  LIN {X 1499.916,Y -481.788,Z -133.994,A 92.55766,B 0.00000,C 180.00000} ; insert
  LIN {X 1499.916,Y -481.788,Z -133.994,A 92.55766,B 0.00000,C 180.00000} ; release
  LIN {X 1499.916,Y -481.788,Z 166.006,A 92.55766,B 0.00000,C 180.00000} ; retreat
  ; Step 2458, bar 2905
  LIN {X 2249.916,Y -481.788,Z 1074.491,A 92.55766,B 0.00000,C 180.00000} ; outside
  LIN {X 2249.916,Y -481.788,Z 116.006,A 92.55766,B 0.00000,C 180.00000} ; preinsert
  LIN {X 2249.916,Y -481.788,Z -133.994,A 92.55766,B 0.00000,C 180.00000} ; insert
  LIN {X 2249.916,Y -481.788,Z -133.994,A 92.55766,B 0.00000,C 180.00000} ; release
  LIN {X 2249.916,Y -481.788,Z 166.006,A 92.55766,B 0.00000,C 180.00000} ; retreat
  ; Step 2459, bar 2908
  LIN {X 2999.916,Y -481.788,Z 1074.491,A 92.55766,B 0.00000,C 180.00000} ; outside
  LIN {X 2999.916,Y -481.788,Z 116.006,A 92.55766,B 0.00000,C 180.00000} ; preinsert
  LIN {X 2999.916,Y -481.788,Z -133.994,A 92.55766,B 0.00000,C 180.00000} ; insert
  LIN {X 2999.916,Y -481.788,Z -133.994,A 92.55766,B 0.00000,C 180.00000} ; release
  LIN {X 2999.916,Y -481.788,Z 166.006,A 92.55766,B 0.00000,C 180.00000} ; retreat
  ; Step 2460, bar 2911
  LIN {X 3749.916,Y -481.788,Z 1074.491,A 92.55766,B 0.00000,C 180.00000} ; outside
  LIN {X 3749.916,Y -481.788,Z 116.006,A 92.55766,B 0.00000,C 180.00000} ; preinsert
  LIN {X 3749.916,Y -481.788,Z -133.994,A 92.55766,B 0.00000,C 180.00000} ; insert
  LIN {X 3749.916,Y -481.788,Z -133.994,A 92.55766,B 0.00000,C 180.00000} ; release
  LIN {X 3749.916,Y -481.788,Z 166.006,A 92.55766,B 0.00000,C 180.00000} ; retreat
  ; Step 2461, bar 2914
  LIN {X 4499.916,Y -481.788,Z 1074.491,A 92.55766,B 0.00000,C 180.00000} ; outside
  LIN {X 4499.916,Y -481.788,Z 116.006,A 92.55766,B 0.00000,C 180.00000} ; preinsert
  LIN {X 4499.916,Y -481.788,Z -133.994,A 92.55766,B 0.00000,C 180.00000} ; insert
  LIN {X 4499.916,Y -481.788,Z -133.994,A 92.55766,B 0.00000,C 180.00000} ; release
  LIN {X 4499.916,Y -481.788,Z 166.006,A 92.55766,B 0.00000,C 180.00000} ; retreat
  ; Step 2462, bar 2917
  LIN {X 5249.916,Y -481.788,Z 1074.491,A 92.55766,B 0.00000,C 180.00000} ; outside
  LIN {X 5249.916,Y -481.788,Z 116.006,A 92.55766,B 0.00000,C 180.00000} ; preinsert
  LIN {X 5249.916,Y -481.788,Z -133.994,A 92.55766,B 0.00000,C 180.00000} ; insert
  LIN {X 5249.916,Y -481.788,Z -133.994,A 92.55766,B 0.00000,C 180.00000} ; release
  LIN {X 5249.916,Y -481.788,Z 166.006,A 92.55766,B 0.00000,C 180.00000} ; retreat
  ; Step 2463, bar 2920
  LIN {X 5999.916,Y -481.788,Z 1074.491,A 92.55766,B 0.00000,C 180.00000} ; outside
  LIN {X 5999.916,Y -481.788,Z 116.006,A 92.55766,B 0.00000,C 180.00000} ; preinsert
  LIN {X 5999.916,Y -481.788,Z -133.994,A 92.55766,B 0.00000,C 180.00000} ; insert
  LIN {X 5999.916,Y -481.788,Z -133.994,A 92.55766,B 0.00000,C 180.00000} ; release
  LIN {X 5999.916,Y -481.788,Z 166.006,A 92.55766,B 0.00000,C 180.00000} ; retreat
  ; Step 2464, bar 2923
  LIN {X 6749.916,Y -481.788,Z 1074.491,A 92.55766,B 0.00000,C 180.00000} ; outside
  LIN {X 6749.916,Y -481.788,Z 116.006,A 92.55766,B 0.00000,C 180.00000} ; preinsert
  LIN {X 6749.916,Y -481.788,Z -133.994,A 92.55766,B 0.00000,C 180.00000} ; insert
  LIN {X 6749.916,Y -481.788,Z -133.994,A 92.55766,B 0.00000,C 180.00000} ; release
  LIN {X 6749.916,Y -481.788,Z 166.006,A 92.55766,B 0.00000,C 180.00000} ; retreat
  ; Step 2465, bar 2926
  LIN {X 7499.916,Y -481.788,Z 1074.491,A 92.55766,B 0.00000,C 180.00000} ; outside
  LIN {X 7499.916,Y -481.788,Z 116.006,A 92.55766,B 0.00000,C 180.00000} ; preinsert
  LIN {X 7499.916,Y -481.788,Z -133.994,A 92.55766,B 0.00000,C 180.00000} ; insert
  LIN {X 7499.916,Y -481.788,Z -133.994,A 92.55766,B 0.00000,C 180.00000} ; release
  LIN {X 7499.916,Y -481.788,Z 166.006,A 92.55766,B 0.00000,C 180.00000} ; retreat
  ; Step 2466, bar 2929
  LIN {X 8249.916,Y -481.788,Z 1074.491,A 92.55766,B 0.00000,C 180.00000} ; outside
  LIN {X 8249.916,Y -481.788,Z 116.006,A 92.55766,B 0.00000,C 180.00000} ; preinsert
  LIN {X 8249.916,Y -481.788,Z -133.994,A 92.55766,B 0.00000,C 180.00000} ; insert
  LIN {X 8249.916,Y -481.788,Z -133.994,A 92.55766,B 0.00000,C 180.00000} ; release
  LIN {X 8249.916,Y -481.788,Z 166.006,A 92.55766,B 0.00000,C 180.00000} ; retreat
  ; Step 2467, bar 2932
  LIN {X 8999.916,Y -481.788,Z 1074.491,A 92.55766,B 0.00000,C 180.00000} ; outside
  LIN {X 8999.916,Y -481.788,Z 116.006,A 92.55766,B 0.00000,C 180.00000} ; preinsert
  LIN {X 8999.916,Y -481.788,Z -133.994,A 92.55766,B 0.00000,C 180.00000} ; insert
  LIN {X 8999.916,Y -481.788,Z -133.994,A 92.55766,B 0.00000,C 180.00000} ; release
  LIN {X 8999.916,Y -481.788,Z 166.006,A 92.55766,B 0.00000,C 180.00000} ; retreat
  ; Step 2468, bar 2935
  LIN {X 9749.916,Y -481.788,Z 1074.491,A 92.55766,B 0.00000,C 180.00000} ; outside
  LIN {X 9749.916,Y -481.788,Z 116.006,A 92.55766,B 0.00000,C 180.00000} ; preinsert
  LIN {X 9749.916,Y -481.788,Z -133.994,A 92.55766,B 0.00000,C 180.00000} ; insert
  LIN {X 9749.916,Y -481.788,Z -133.994,A 92.55766,B 0.00000,C 180.00000} ; release
  LIN {X 9749.916,Y -481.788,Z 166.006,A 92.55766,B 0.00000,C 180.00000} ; retreat
  ; Step 2469, bar 2938
  LIN {X 10499.916,Y -481.788,Z 1074.491,A 92.55766,B 0.00000,C 180.00000} ; outside
  LIN {X 10499.916,Y -481.788,Z 116.006,A 92.55766,B 0.00000,C 180.00000} ; preinsert
  LIN {X 10499.916,Y -481.788,Z -133.994,A 92.55766,B 0.00000,C 180.00000} ; insert
  LIN {X 10499.916,Y -481.788,Z -133.994,A 92.55766,B 0.00000,C 180.00000} ; release
  LIN {X 10499.916,Y -481.788,Z 166.006,A 92.55766,B 0.00000,C 180.00000} ; retreat
  ; Step 2470, bar 2941
  LIN {X 11249.916,Y -481.788,Z 1074.491,A 92.55766,B 0.00000,C 180.00000} ; outside
  LIN {X 11249.916,Y -481.788,Z 116.006,A 92.55766,B 0.00000,C 180.00000} ; preinsert
  LIN {X 11249.916,Y -481.788,Z -133.994,A 92.55766,B 0.00000,C 180.00000} ; insert
  LIN {X 11249.916,Y -481.788,Z -133.994,A 92.55766,B 0.00000,C 180.00000} ; release
  LIN {X 11249.916,Y -481.788,Z 166.006,A 92.55766,B 0.00000,C 180.00000} ; retreat
  ; Step 2471, bar 2943
  LIN {X 11999.916,Y -481.788,Z 1074.491,A 92.55766,B 0.00000,C 180.00000} ; outside
  LIN {X 11999.916,Y -481.788,Z 116.006,A 92.55766,B 0.00000,C 180.00000} ; preinsert
  LIN {X 11999.916,Y -481.788,Z -133.994,A 92.55766,B 0.00000,C 180.00000} ; insert
  LIN {X 11999.916,Y -481.788,Z -133.994,A 92.55766,B 0.00000,C 180.00000} ; release
  LIN {X 11999.916,Y -481.788,Z 166.006,A 92.55766,B 0.00000,C 180.00000} ; retreat
  ; Step 2472, bar 2636
  LIN {X -11999.916,Y 481.788,Z 1074.491,A -87.44234,B 0.00000,C 180.00000} ; outside
  LIN {X -11999.916,Y 481.788,Z 116.006,A -87.44234,B 0.00000,C 180.00000} ; preinsert
  LIN {X -11999.916,Y 481.788,Z -133.994,A -87.44234,B 0.00000,C 180.00000} ; insert
  LIN {X -11999.916,Y 481.788,Z -133.994,A -87.44234,B 0.00000,C 180.00000} ; release
  LIN {X -11999.916,Y 481.788,Z 166.006,A -87.44234,B 0.00000,C 180.00000} ; retreat
  ; Step 2473, bar 2631
  LIN {X -11249.916,Y 481.788,Z 1074.491,A -87.44234,B 0.00000,C 180.00000} ; outside
  LIN {X -11249.916,Y 481.788,Z 116.006,A -87.44234,B 0.00000,C 180.00000} ; preinsert
  LIN {X -11249.916,Y 481.788,Z -133.994,A -87.44234,B 0.00000,C 180.00000} ; insert
  LIN {X -11249.916,Y 481.788,Z -133.994,A -87.44234,B 0.00000,C 180.00000} ; release
  LIN {X -11249.916,Y 481.788,Z 166.006,A -87.44234,B 0.00000,C 180.00000} ; retreat
  ; Step 2474, bar 2624
  LIN {X -10499.916,Y 481.788,Z 1074.491,A -87.44234,B 0.00000,C 180.00000} ; outside
  LIN {X -10499.916,Y 481.788,Z 116.006,A -87.44234,B 0.00000,C 180.00000} ; preinsert
  LIN {X -10499.916,Y 481.788,Z -133.994,A -87.44234,B 0.00000,C 180.00000} ; insert
  LIN {X -10499.916,Y 481.788,Z -133.994,A -87.44234,B 0.00000,C 180.00000} ; release
  LIN {X -10499.916,Y 481.788,Z 166.006,A -87.44234,B 0.00000,C 180.00000} ; retreat
  ; Step 2475, bar 2617
  LIN {X -9749.916,Y 481.788,Z 1074.491,A -87.44234,B 0.00000,C 180.00000} ; outside
  LIN {X -9749.916,Y 481.788,Z 116.006,A -87.44234,B 0.00000,C 180.00000} ; preinsert
  LIN {X -9749.916,Y 481.788,Z -133.994,A -87.44234,B 0.00000,C 180.00000} ; insert
  LIN {X -9749.916,Y 481.788,Z -133.994,A -87.44234,B 0.00000,C 180.00000} ; release
  LIN {X -9749.916,Y 481.788,Z 166.006,A -87.44234,B 0.00000,C 180.00000} ; retreat
  ; Step 2476, bar 2610
  LIN {X -8999.916,Y 481.788,Z 1074.491,A -87.44234,B 0.00000,C 180.00000} ; outside
  LIN {X -8999.916,Y 481.788,Z 116.006,A -87.44234,B 0.00000,C 180.00000} ; preinsert
  LIN {X -8999.916,Y 481.788,Z -133.994,A -87.44234,B 0.00000,C 180.00000} ; insert
  LIN {X -8999.916,Y 481.788,Z -133.994,A -87.44234,B 0.00000,C 180.00000} ; release
  LIN {X -8999.916,Y 481.788,Z 166.006,A -87.44234,B 0.00000,C 180.00000} ; retreat
  ; Step 2477, bar 2603
  LIN {X -8249.916,Y 481.788,Z 1074.491,A -87.44234,B 0.00000,C 180.00000} ; outside
  LIN {X -8249.916,Y 481.788,Z 116.006,A -87.44234,B 0.00000,C 180.00000} ; preinsert
  LIN {X -8249.916,Y 481.788,Z -133.994,A -87.44234,B 0.00000,C 180.00000} ; insert
  LIN {X -8249.916,Y 481.788,Z -133.994,A -87.44234,B 0.00000,C 180.00000} ; release
  LIN {X -8249.916,Y 481.788,Z 166.006,A -87.44234,B 0.00000,C 180.00000} ; retreat
  ; Step 2478, bar 2596
  LIN {X -7499.916,Y 481.788,Z 1074.491,A -87.44234,B 0.00000,C 180.00000} ; outside
  LIN {X -7499.916,Y 481.788,Z 116.006,A -87.44234,B 0.00000,C 180.00000} ; preinsert
  LIN {X -7499.916,Y 481.788,Z -133.994,A -87.44234,B 0.00000,C 180.00000} ; insert
  LIN {X -7499.916,Y 481.788,Z -133.994,A -87.44234,B 0.00000,C 180.00000} ; release
  LIN {X -7499.916,Y 481.788,Z 166.006,A -87.44234,B 0.00000,C 180.00000} ; retreat
  ; Step 2479, bar 2589
  LIN {X -6749.916,Y 481.788,Z 1074.491,A -87.44234,B 0.00000,C 180.00000} ; outside
  LIN {X -6749.916,Y 481.788,Z 116.006,A -87.44234,B 0.00000,C 180.00000} ; preinsert
  LIN {X -6749.916,Y 481.788,Z -133.994,A -87.44234,B 0.00000,C 180.00000} ; insert
  LIN {X -6749.916,Y 481.788,Z -133.994,A -87.44234,B 0.00000,C 180.00000} ; release
  LIN {X -6749.916,Y 481.788,Z 166.006,A -87.44234,B 0.00000,C 180.00000} ; retreat
  ; Step 2480, bar 2582
  LIN {X -5999.916,Y 481.788,Z 1074.491,A -87.44234,B 0.00000,C 180.00000} ; outside
  LIN {X -5999.916,Y 481.788,Z 116.006,A -87.44234,B 0.00000,C 180.00000} ; preinsert
  LIN {X -5999.916,Y 481.788,Z -133.994,A -87.44234,B 0.00000,C 180.00000} ; insert
  LIN {X -5999.916,Y 481.788,Z -133.994,A -87.44234,B 0.00000,C 180.00000} ; release
  LIN {X -5999.916,Y 481.788,Z 166.006,A -87.44234,B 0.00000,C 180.00000} ; retreat
  ; Step 2481, bar 2575
  LIN {X -5249.916,Y 481.788,Z 1074.491,A -87.44234,B 0.00000,C 180.00000} ; outside
  LIN {X -5249.916,Y 481.788,Z 116.006,A -87.44234,B 0.00000,C 180.00000} ; preinsert
  LIN {X -5249.916,Y 481.788,Z -133.994,A -87.44234,B 0.00000,C 180.00000} ; insert
  LIN {X -5249.916,Y 481.788,Z -133.994,A -87.44234,B 0.00000,C 180.00000} ; release
  LIN {X -5249.916,Y 481.788,Z 166.006,A -87.44234,B 0.00000,C 180.00000} ; retreat
  ; Step 2482, bar 2568
  LIN {X -4499.916,Y 481.788,Z 1074.491,A -87.44234,B 0.00000,C 180.00000} ; outside
  LIN {X -4499.916,Y 481.788,Z 116.006,A -87.44234,B 0.00000,C 180.00000} ; preinsert
  LIN {X -4499.916,Y 481.788,Z -133.994,A -87.44234,B 0.00000,C 180.00000} ; insert
  LIN {X -4499.916,Y 481.788,Z -133.994,A -87.44234,B 0.00000,C 180.00000} ; release
  LIN {X -4499.916,Y 481.788,Z 166.006,A -87.44234,B 0.00000,C 180.00000} ; retreat
  ; Step 2483, bar 2561
  LIN {X -3749.916,Y 481.788,Z 1074.491,A -87.44234,B 0.00000,C 180.00000} ; outside
  LIN {X -3749.916,Y 481.788,Z 116.006,A -87.44234,B 0.00000,C 180.00000} ; preinsert
  LIN {X -3749.916,Y 481.788,Z -133.994,A -87.44234,B 0.00000,C 180.00000} ; insert
  LIN {X -3749.916,Y 481.788,Z -133.994,A -87.44234,B 0.00000,C 180.00000} ; release
  LIN {X -3749.916,Y 481.788,Z 166.006,A -87.44234,B 0.00000,C 180.00000} ; retreat
  ; Step 2484, bar 2554
  LIN {X -2999.916,Y 481.788,Z 1074.491,A -87.44234,B 0.00000,C 180.00000} ; outside
  LIN {X -2999.916,Y 481.788,Z 116.006,A -87.44234,B 0.00000,C 180.00000} ; preinsert
  LIN {X -2999.916,Y 481.788,Z -133.994,A -87.44234,B 0.00000,C 180.00000} ; insert
  LIN {X -2999.916,Y 481.788,Z -133.994,A -87.44234,B 0.00000,C 180.00000} ; release
  LIN {X -2999.916,Y 481.788,Z 166.006,A -87.44234,B 0.00000,C 180.00000} ; retreat
  ; Step 2485, bar 2547
  LIN {X -2249.916,Y 481.788,Z 1074.491,A -87.44234,B 0.00000,C 180.00000} ; outside
  LIN {X -2249.916,Y 481.788,Z 116.006,A -87.44234,B 0.00000,C 180.00000} ; preinsert
  LIN {X -2249.916,Y 481.788,Z -133.994,A -87.44234,B 0.00000,C 180.00000} ; insert
  LIN {X -2249.916,Y 481.788,Z -133.994,A -87.44234,B 0.00000,C 180.00000} ; release
  LIN {X -2249.916,Y 481.788,Z 166.006,A -87.44234,B 0.00000,C 180.00000} ; retreat
  ; Step 2486, bar 2540
  LIN {X -1499.916,Y 481.788,Z 1074.491,A -87.44234,B 0.00000,C 180.00000} ; outside
  LIN {X -1499.916,Y 481.788,Z 116.006,A -87.44234,B 0.00000,C 180.00000} ; preinsert
  LIN {X -1499.916,Y 481.788,Z -133.994,A -87.44234,B 0.00000,C 180.00000} ; insert
  LIN {X -1499.916,Y 481.788,Z -133.994,A -87.44234,B 0.00000,C 180.00000} ; release
  LIN {X -1499.916,Y 481.788,Z 166.006,A -87.44234,B 0.00000,C 180.00000} ; retreat
  ; Step 2487, bar 1974
  LIN {X 0.084,Y 481.788,Z 1074.491,A -87.44234,B 0.00000,C 180.00000} ; outside
  LIN {X 0.084,Y 481.788,Z 116.006,A -87.44234,B 0.00000,C 180.00000} ; preinsert
  LIN {X 0.084,Y 481.788,Z -133.994,A -87.44234,B 0.00000,C 180.00000} ; insert
  LIN {X 0.084,Y 481.788,Z -133.994,A -87.44234,B 0.00000,C 180.00000} ; release
  LIN {X 0.084,Y 481.788,Z 166.006,A -87.44234,B 0.00000,C 180.00000} ; retreat
  ; Step 2488, bar 2693
  LIN {X 1499.916,Y 481.788,Z 1074.491,A -92.55766,B 0.00000,C -180.00000} ; outside
  LIN {X 1499.916,Y 481.788,Z 116.006,A -92.55766,B 0.00000,C -180.00000} ; preinsert
  LIN {X 1499.916,Y 481.788,Z -133.994,A -92.55766,B 0.00000,C -180.00000} ; insert
  LIN {X 1499.916,Y 481.788,Z -133.994,A -92.55766,B 0.00000,C -180.00000} ; release
  LIN {X 1499.916,Y 481.788,Z 166.006,A -92.55766,B 0.00000,C -180.00000} ; retreat
  ; Step 2489, bar 2697
  LIN {X 2249.916,Y 481.788,Z 1074.491,A -92.55766,B 0.00000,C -180.00000} ; outside
  LIN {X 2249.916,Y 481.788,Z 116.006,A -92.55766,B 0.00000,C -180.00000} ; preinsert
  LIN {X 2249.916,Y 481.788,Z -133.994,A -92.55766,B 0.00000,C -180.00000} ; insert
  LIN {X 2249.916,Y 481.788,Z -133.994,A -92.55766,B 0.00000,C -180.00000} ; release
  LIN {X 2249.916,Y 481.788,Z 166.006,A -92.55766,B 0.00000,C -180.00000} ; retreat
  ; Step 2490, bar 2701
  LIN {X 2999.916,Y 481.788,Z 1074.491,A -92.55766,B 0.00000,C -180.00000} ; outside
  LIN {X 2999.916,Y 481.788,Z 116.006,A -92.55766,B 0.00000,C -180.00000} ; preinsert
  LIN {X 2999.916,Y 481.788,Z -133.994,A -92.55766,B 0.00000,C -180.00000} ; insert
  LIN {X 2999.916,Y 481.788,Z -133.994,A -92.55766,B 0.00000,C -180.00000} ; release
  LIN {X 2999.916,Y 481.788,Z 166.006,A -92.55766,B 0.00000,C -180.00000} ; retreat
  ; Step 2491, bar 2705
  LIN {X 3749.916,Y 481.788,Z 1074.491,A -92.55766,B 0.00000,C -180.00000} ; outside
  LIN {X 3749.916,Y 481.788,Z 116.006,A -92.55766,B 0.00000,C -180.00000} ; preinsert
  LIN {X 3749.916,Y 481.788,Z -133.994,A -92.55766,B 0.00000,C -180.00000} ; insert
  LIN {X 3749.916,Y 481.788,Z -133.994,A -92.55766,B 0.00000,C -180.00000} ; release
  LIN {X 3749.916,Y 481.788,Z 166.006,A -92.55766,B 0.00000,C -180.00000} ; retreat
  ; Step 2492, bar 2709
  LIN {X 4499.916,Y 481.788,Z 1074.491,A -92.55766,B 0.00000,C -180.00000} ; outside
  LIN {X 4499.916,Y 481.788,Z 116.006,A -92.55766,B 0.00000,C -180.00000} ; preinsert
  LIN {X 4499.916,Y 481.788,Z -133.994,A -92.55766,B 0.00000,C -180.00000} ; insert
  LIN {X 4499.916,Y 481.788,Z -133.994,A -92.55766,B 0.00000,C -180.00000} ; release
  LIN {X 4499.916,Y 481.788,Z 166.006,A -92.55766,B 0.00000,C -180.00000} ; retreat
  ; Step 2493, bar 2713
  LIN {X 5249.916,Y 481.788,Z 1074.491,A -92.55766,B 0.00000,C -180.00000} ; outside
  LIN {X 5249.916,Y 481.788,Z 116.006,A -92.55766,B 0.00000,C -180.00000} ; preinsert
  LIN {X 5249.916,Y 481.788,Z -133.994,A -92.55766,B 0.00000,C -180.00000} ; insert
  LIN {X 5249.916,Y 481.788,Z -133.994,A -92.55766,B 0.00000,C -180.00000} ; release
  LIN {X 5249.916,Y 481.788,Z 166.006,A -92.55766,B 0.00000,C -180.00000} ; retreat
  ; Step 2494, bar 2717
  LIN {X 5999.916,Y 481.788,Z 1074.491,A -92.55766,B 0.00000,C -180.00000} ; outside
  LIN {X 5999.916,Y 481.788,Z 116.006,A -92.55766,B 0.00000,C -180.00000} ; preinsert
  LIN {X 5999.916,Y 481.788,Z -133.994,A -92.55766,B 0.00000,C -180.00000} ; insert
  LIN {X 5999.916,Y 481.788,Z -133.994,A -92.55766,B 0.00000,C -180.00000} ; release
  LIN {X 5999.916,Y 481.788,Z 166.006,A -92.55766,B 0.00000,C -180.00000} ; retreat
  ; Step 2495, bar 2721
  LIN {X 6749.916,Y 481.788,Z 1074.491,A -92.55766,B 0.00000,C -180.00000} ; outside
  LIN {X 6749.916,Y 481.788,Z 116.006,A -92.55766,B 0.00000,C -180.00000} ; preinsert
  LIN {X 6749.916,Y 481.788,Z -133.994,A -92.55766,B 0.00000,C -180.00000} ; insert
  LIN {X 6749.916,Y 481.788,Z -133.994,A -92.55766,B 0.00000,C -180.00000} ; release
  LIN {X 6749.916,Y 481.788,Z 166.006,A -92.55766,B 0.00000,C -180.00000} ; retreat
  ; Step 2496, bar 2725
  LIN {X 7499.916,Y 481.788,Z 1074.491,A -92.55766,B 0.00000,C -180.00000} ; outside
  LIN {X 7499.916,Y 481.788,Z 116.006,A -92.55766,B 0.00000,C -180.00000} ; preinsert
  LIN {X 7499.916,Y 481.788,Z -133.994,A -92.55766,B 0.00000,C -180.00000} ; insert
  LIN {X 7499.916,Y 481.788,Z -133.994,A -92.55766,B 0.00000,C -180.00000} ; release
  LIN {X 7499.916,Y 481.788,Z 166.006,A -92.55766,B 0.00000,C -180.00000} ; retreat
  ; Step 2497, bar 2729
  LIN {X 8249.916,Y 481.788,Z 1074.491,A -92.55766,B 0.00000,C -180.00000} ; outside
  LIN {X 8249.916,Y 481.788,Z 116.006,A -92.55766,B 0.00000,C -180.00000} ; preinsert
  LIN {X 8249.916,Y 481.788,Z -133.994,A -92.55766,B 0.00000,C -180.00000} ; insert
  LIN {X 8249.916,Y 481.788,Z -133.994,A -92.55766,B 0.00000,C -180.00000} ; release
  LIN {X 8249.916,Y 481.788,Z 166.006,A -92.55766,B 0.00000,C -180.00000} ; retreat
  ; Step 2498, bar 2733
  LIN {X 8999.916,Y 481.788,Z 1074.491,A -92.55766,B 0.00000,C -180.00000} ; outside
  LIN {X 8999.916,Y 481.788,Z 116.006,A -92.55766,B 0.00000,C -180.00000} ; preinsert
  LIN {X 8999.916,Y 481.788,Z -133.994,A -92.55766,B 0.00000,C -180.00000} ; insert
  LIN {X 8999.916,Y 481.788,Z -133.994,A -92.55766,B 0.00000,C -180.00000} ; release
  LIN {X 8999.916,Y 481.788,Z 166.006,A -92.55766,B 0.00000,C -180.00000} ; retreat
  ; Step 2499, bar 2737
  LIN {X 9749.916,Y 481.788,Z 1074.491,A -92.55766,B 0.00000,C -180.00000} ; outside
  LIN {X 9749.916,Y 481.788,Z 116.006,A -92.55766,B 0.00000,C -180.00000} ; preinsert
  LIN {X 9749.916,Y 481.788,Z -133.994,A -92.55766,B 0.00000,C -180.00000} ; insert
  LIN {X 9749.916,Y 481.788,Z -133.994,A -92.55766,B 0.00000,C -180.00000} ; release
  LIN {X 9749.916,Y 481.788,Z 166.006,A -92.55766,B 0.00000,C -180.00000} ; retreat
  ; Step 2500, bar 2741
  LIN {X 10499.916,Y 481.788,Z 1074.491,A -92.55766,B 0.00000,C -180.00000} ; outside
  LIN {X 10499.916,Y 481.788,Z 116.006,A -92.55766,B 0.00000,C -180.00000} ; preinsert
  LIN {X 10499.916,Y 481.788,Z -133.994,A -92.55766,B 0.00000,C -180.00000} ; insert
  LIN {X 10499.916,Y 481.788,Z -133.994,A -92.55766,B 0.00000,C -180.00000} ; release
  LIN {X 10499.916,Y 481.788,Z 166.006,A -92.55766,B 0.00000,C -180.00000} ; retreat
  ; Step 2501, bar 2745
  LIN {X 11249.916,Y 481.788,Z 1074.491,A -92.55766,B 0.00000,C -180.00000} ; outside
  LIN {X 11249.916,Y 481.788,Z 116.006,A -92.55766,B 0.00000,C -180.00000} ; preinsert
  LIN {X 11249.916,Y 481.788,Z -133.994,A -92.55766,B 0.00000,C -180.00000} ; insert
  LIN {X 11249.916,Y 481.788,Z -133.994,A -92.55766,B 0.00000,C -180.00000} ; release
  LIN {X 11249.916,Y 481.788,Z 166.006,A -92.55766,B 0.00000,C -180.00000} ; retreat
  ; Step 2502, bar 2748
  LIN {X 11999.916,Y 481.788,Z 1074.491,A -92.55766,B 0.00000,C -180.00000} ; outside
  LIN {X 11999.916,Y 481.788,Z 116.006,A -92.55766,B 0.00000,C -180.00000} ; preinsert
  LIN {X 11999.916,Y 481.788,Z -133.994,A -92.55766,B 0.00000,C -180.00000} ; insert
  LIN {X 11999.916,Y 481.788,Z -133.994,A -92.55766,B 0.00000,C -180.00000} ; release
  LIN {X 11999.916,Y 481.788,Z 166.006,A -92.55766,B 0.00000,C -180.00000} ; retreat
  ; Step 2503, bar 2533
  LIN {X -749.916,Y 481.788,Z 1074.491,A -87.44234,B 0.00000,C -180.00000} ; outside
  LIN {X -749.916,Y 481.788,Z 116.006,A -87.44234,B 0.00000,C -180.00000} ; preinsert
  LIN {X -749.916,Y 481.788,Z -133.994,A -87.44234,B 0.00000,C -180.00000} ; insert
  LIN {X -749.916,Y 481.788,Z -133.994,A -87.44234,B 0.00000,C -180.00000} ; release
  LIN {X -749.916,Y 481.788,Z 166.006,A -87.44234,B 0.00000,C -180.00000} ; retreat
  ; Step 2504, bar 2689
  LIN {X 749.916,Y 481.788,Z 1074.491,A -92.55766,B 0.00000,C -180.00000} ; outside
  LIN {X 749.916,Y 481.788,Z 116.006,A -92.55766,B 0.00000,C -180.00000} ; preinsert
  LIN {X 749.916,Y 481.788,Z -133.994,A -92.55766,B 0.00000,C -180.00000} ; insert
  LIN {X 749.916,Y 481.788,Z -133.994,A -92.55766,B 0.00000,C -180.00000} ; release
  LIN {X 749.916,Y 481.788,Z 166.006,A -92.55766,B 0.00000,C -180.00000} ; retreat
  ; Step 2505, bar 2979
  LIN {X -14850.033,Y -731.601,Z 992.718,A 131.29142,B 0.00000,C -180.00000} ; outside
  LIN {X -14850.033,Y -731.601,Z 31.921,A 131.29142,B 0.00000,C -180.00000} ; preinsert
  LIN {X -14850.033,Y -731.601,Z -218.079,A 131.29142,B 0.00000,C -180.00000} ; insert
  LIN {X -14850.033,Y -731.601,Z -218.079,A 131.29142,B 0.00000,C -180.00000} ; release
  LIN {X -14850.033,Y -731.601,Z 81.921,A 131.29142,B 0.00000,C -180.00000} ; retreat
  ; Step 2506, bar 3000
  LIN {X 14850.033,Y 731.601,Z 992.718,A -48.70858,B 0.00000,C 180.00000} ; outside
  LIN {X 14850.033,Y 731.601,Z 31.921,A -48.70858,B 0.00000,C 180.00000} ; preinsert
  LIN {X 14850.033,Y 731.601,Z -218.079,A -48.70858,B 0.00000,C 180.00000} ; insert
  LIN {X 14850.033,Y 731.601,Z -218.079,A -48.70858,B 0.00000,C 180.00000} ; release
  LIN {X 14850.033,Y 731.601,Z 81.921,A -48.70858,B 0.00000,C 180.00000} ; retreat
  ; Step 2507, bar 3018
  LIN {X 14850.033,Y -731.601,Z 992.718,A 48.70858,B 0.00000,C 180.00000} ; outside
  LIN {X 14850.033,Y -731.601,Z 31.920,A 48.70858,B 0.00000,C 180.00000} ; preinsert
  LIN {X 14850.033,Y -731.601,Z -218.080,A 48.70858,B 0.00000,C 180.00000} ; insert
  LIN {X 14850.033,Y -731.601,Z -218.080,A 48.70858,B 0.00000,C 180.00000} ; release
  LIN {X 14850.033,Y -731.601,Z 81.920,A 48.70858,B 0.00000,C 180.00000} ; retreat
  ; Step 2508, bar 2961
  LIN {X -14850.033,Y 731.601,Z 992.718,A -131.29142,B 0.00000,C 180.00000} ; outside
  LIN {X -14850.033,Y 731.601,Z 31.920,A -131.29142,B 0.00000,C 180.00000} ; preinsert
  LIN {X -14850.033,Y 731.601,Z -218.080,A -131.29142,B 0.00000,C 180.00000} ; insert
  LIN {X -14850.033,Y 731.601,Z -218.080,A -131.29142,B 0.00000,C 180.00000} ; release
  LIN {X -14850.033,Y 731.601,Z 81.920,A -131.29142,B 0.00000,C 180.00000} ; retreat
  ; Step 2509, bar 3015
  LIN {X 14450.033,Y -481.600,Z 1007.193,A 48.70858,B 0.00000,C 180.00000} ; outside
  LIN {X 14450.033,Y -481.600,Z 46.708,A 48.70858,B 0.00000,C 180.00000} ; preinsert
  LIN {X 14450.033,Y -481.600,Z -203.292,A 48.70858,B 0.00000,C 180.00000} ; insert
  LIN {X 14450.033,Y -481.600,Z -203.292,A 48.70858,B 0.00000,C 180.00000} ; release
  LIN {X 14450.033,Y -481.600,Z 96.708,A 48.70858,B 0.00000,C 180.00000} ; retreat
  ; Step 2510, bar 2958
  LIN {X -14450.033,Y 481.600,Z 1007.193,A -131.29142,B 0.00000,C -180.00000} ; outside
  LIN {X -14450.033,Y 481.600,Z 46.708,A -131.29142,B 0.00000,C -180.00000} ; preinsert
  LIN {X -14450.033,Y 481.600,Z -203.292,A -131.29142,B 0.00000,C -180.00000} ; insert
  LIN {X -14450.033,Y 481.600,Z -203.292,A -131.29142,B 0.00000,C -180.00000} ; release
  LIN {X -14450.033,Y 481.600,Z 96.708,A -131.29142,B 0.00000,C -180.00000} ; retreat
  ; Step 2511, bar 2976
  LIN {X -14450.033,Y -481.600,Z 1007.193,A 131.29142,B 0.00000,C -180.00000} ; outside
  LIN {X -14450.033,Y -481.600,Z 46.709,A 131.29142,B 0.00000,C -180.00000} ; preinsert
  LIN {X -14450.033,Y -481.600,Z -203.291,A 131.29142,B 0.00000,C -180.00000} ; insert
  LIN {X -14450.033,Y -481.600,Z -203.291,A 131.29142,B 0.00000,C -180.00000} ; release
  LIN {X -14450.033,Y -481.600,Z 96.709,A 131.29142,B 0.00000,C -180.00000} ; retreat
  ; Step 2512, bar 2997
  LIN {X 14450.033,Y 481.600,Z 1007.193,A -48.70858,B 0.00000,C 180.00000} ; outside
  LIN {X 14450.033,Y 481.600,Z 46.709,A -48.70858,B 0.00000,C 180.00000} ; preinsert
  LIN {X 14450.033,Y 481.600,Z -203.291,A -48.70858,B 0.00000,C 180.00000} ; insert
  LIN {X 14450.033,Y 481.600,Z -203.291,A -48.70858,B 0.00000,C 180.00000} ; release
  LIN {X 14450.033,Y 481.600,Z 96.709,A -48.70858,B 0.00000,C 180.00000} ; retreat
  ; Step 2513, bar 3013
  LIN {X 14050.033,Y -731.600,Z 1011.349,A 48.70858,B 0.00000,C 180.00000} ; outside
  LIN {X 14050.033,Y -731.600,Z 50.552,A 48.70858,B 0.00000,C 180.00000} ; preinsert
  LIN {X 14050.033,Y -731.600,Z -199.448,A 48.70858,B 0.00000,C 180.00000} ; insert
  LIN {X 14050.033,Y -731.600,Z -199.448,A 48.70858,B 0.00000,C 180.00000} ; release
  LIN {X 14050.033,Y -731.600,Z 100.552,A 48.70858,B 0.00000,C 180.00000} ; retreat
  ; Step 2514, bar 2974
  LIN {X -14050.033,Y -731.600,Z 1011.349,A 131.29142,B 0.00000,C 180.00000} ; outside
  LIN {X -14050.033,Y -731.600,Z 50.552,A 131.29142,B 0.00000,C 180.00000} ; preinsert
  LIN {X -14050.033,Y -731.600,Z -199.448,A 131.29142,B 0.00000,C 180.00000} ; insert
  LIN {X -14050.033,Y -731.600,Z -199.448,A 131.29142,B 0.00000,C 180.00000} ; release
  LIN {X -14050.033,Y -731.600,Z 100.552,A 131.29142,B 0.00000,C 180.00000} ; retreat
  ; Step 2515, bar 2955
  LIN {X -14050.033,Y 731.600,Z 1011.349,A -131.29142,B 0.00000,C -180.00000} ; outside
  LIN {X -14050.033,Y 731.600,Z 50.552,A -131.29142,B 0.00000,C -180.00000} ; preinsert
  LIN {X -14050.033,Y 731.600,Z -199.448,A -131.29142,B 0.00000,C -180.00000} ; insert
  LIN {X -14050.033,Y 731.600,Z -199.448,A -131.29142,B 0.00000,C -180.00000} ; release
  LIN {X -14050.033,Y 731.600,Z 100.552,A -131.29142,B 0.00000,C -180.00000} ; retreat
  ; Step 2516, bar 2994
  LIN {X 14050.033,Y 731.600,Z 1011.349,A -48.70858,B 0.00000,C 180.00000} ; outside
  LIN {X 14050.033,Y 731.600,Z 50.552,A -48.70858,B 0.00000,C 180.00000} ; preinsert
  LIN {X 14050.033,Y 731.600,Z -199.448,A -48.70858,B 0.00000,C 180.00000} ; insert
  LIN {X 14050.033,Y 731.600,Z -199.448,A -48.70858,B 0.00000,C 180.00000} ; release
  LIN {X 14050.033,Y 731.600,Z 100.552,A -48.70858,B 0.00000,C 180.00000} ; retreat
  ; Step 2517, bar 3010
  LIN {X 13649.947,Y -481.615,Z 1025.484,A 88.24449,B 0.00000,C 180.00000} ; outside
  LIN {X 13649.947,Y -481.615,Z 64.999,A 88.24449,B 0.00000,C 180.00000} ; preinsert
  LIN {X 13649.947,Y -481.615,Z -185.001,A 88.24449,B 0.00000,C 180.00000} ; insert
  LIN {X 13649.947,Y -481.615,Z -185.001,A 88.24449,B 0.00000,C 180.00000} ; release
  LIN {X 13649.947,Y -481.615,Z 114.999,A 88.24449,B 0.00000,C 180.00000} ; retreat
  ; Step 2518, bar 2952
  LIN {X -13649.947,Y 481.615,Z 1025.484,A -91.75551,B 0.00000,C -180.00000} ; outside
  LIN {X -13649.947,Y 481.615,Z 64.999,A -91.75551,B 0.00000,C -180.00000} ; preinsert
  LIN {X -13649.947,Y 481.615,Z -185.001,A -91.75551,B 0.00000,C -180.00000} ; insert
  LIN {X -13649.947,Y 481.615,Z -185.001,A -91.75551,B 0.00000,C -180.00000} ; release
  LIN {X -13649.947,Y 481.615,Z 114.999,A -91.75551,B 0.00000,C -180.00000} ; retreat
  ; Step 2519, bar 2971
  LIN {X -13649.947,Y -481.615,Z 1025.484,A 91.75551,B 0.00000,C 180.00000} ; outside
  LIN {X -13649.947,Y -481.615,Z 64.999,A 91.75551,B 0.00000,C 180.00000} ; preinsert
  LIN {X -13649.947,Y -481.615,Z -185.001,A 91.75551,B 0.00000,C 180.00000} ; insert
  LIN {X -13649.947,Y -481.615,Z -185.001,A 91.75551,B 0.00000,C 180.00000} ; release
  LIN {X -13649.947,Y -481.615,Z 114.999,A 91.75551,B 0.00000,C 180.00000} ; retreat
  ; Step 2520, bar 2991
  LIN {X 13649.947,Y 481.615,Z 1025.484,A -88.24449,B 0.00000,C 180.00000} ; outside
  LIN {X 13649.947,Y 481.615,Z 64.999,A -88.24449,B 0.00000,C 180.00000} ; preinsert
  LIN {X 13649.947,Y 481.615,Z -185.001,A -88.24449,B 0.00000,C 180.00000} ; insert
  LIN {X 13649.947,Y 481.615,Z -185.001,A -88.24449,B 0.00000,C 180.00000} ; release
  LIN {X 13649.947,Y 481.615,Z 114.999,A -88.24449,B 0.00000,C 180.00000} ; retreat
  ; Step 2521, bar 3008
  LIN {X 13250.050,Y -731.639,Z 1044.389,A 88.44949,B 0.00000,C -180.00000} ; outside
  LIN {X 13250.050,Y -731.639,Z 83.592,A 88.44949,B 0.00000,C -180.00000} ; preinsert
  LIN {X 13250.050,Y -731.639,Z -166.408,A 88.44949,B 0.00000,C -180.00000} ; insert
  LIN {X 13250.050,Y -731.639,Z -166.408,A 88.44949,B 0.00000,C -180.00000} ; release
  LIN {X 13250.050,Y -731.639,Z 133.592,A 88.44949,B 0.00000,C -180.00000} ; retreat
  ; Step 2522, bar 2949
  LIN {X -13250.050,Y 731.639,Z 1044.389,A -91.55051,B 0.00000,C -180.00000} ; outside
  LIN {X -13250.050,Y 731.639,Z 83.592,A -91.55051,B 0.00000,C -180.00000} ; preinsert
  LIN {X -13250.050,Y 731.639,Z -166.408,A -91.55051,B 0.00000,C -180.00000} ; insert
  LIN {X -13250.050,Y 731.639,Z -166.408,A -91.55051,B 0.00000,C -180.00000} ; release
  LIN {X -13250.050,Y 731.639,Z 133.592,A -91.55051,B 0.00000,C -180.00000} ; retreat
  ; Step 2523, bar 2969
  LIN {X -13250.050,Y -731.639,Z 1044.389,A 91.55051,B 0.00000,C 180.00000} ; outside
  LIN {X -13250.050,Y -731.639,Z 83.592,A 91.55051,B 0.00000,C 180.00000} ; preinsert
  LIN {X -13250.050,Y -731.639,Z -166.408,A 91.55051,B 0.00000,C 180.00000} ; insert
  LIN {X -13250.050,Y -731.639,Z -166.408,A 91.55051,B 0.00000,C 180.00000} ; release
  LIN {X -13250.050,Y -731.639,Z 133.592,A 91.55051,B 0.00000,C 180.00000} ; retreat
  ; Step 2524, bar 2988
  LIN {X 13250.050,Y 731.639,Z 1044.389,A -88.44949,B 0.00000,C -180.00000} ; outside
  LIN {X 13250.050,Y 731.639,Z 83.592,A -88.44949,B 0.00000,C -180.00000} ; preinsert
  LIN {X 13250.050,Y 731.639,Z -166.408,A -88.44949,B 0.00000,C -180.00000} ; insert
  LIN {X 13250.050,Y 731.639,Z -166.408,A -88.44949,B 0.00000,C -180.00000} ; release
  LIN {X 13250.050,Y 731.639,Z 133.592,A -88.44949,B 0.00000,C -180.00000} ; retreat
  ; Step 2525, bar 3005
  LIN {X 12850.013,Y -481.830,Z 1050.408,A 89.15631,B 0.00000,C 180.00000} ; outside
  LIN {X 12850.013,Y -481.830,Z 89.924,A 89.15631,B 0.00000,C 180.00000} ; preinsert
  LIN {X 12850.013,Y -481.830,Z -160.076,A 89.15631,B 0.00000,C 180.00000} ; insert
  LIN {X 12850.013,Y -481.830,Z -160.076,A 89.15631,B 0.00000,C 180.00000} ; release
  LIN {X 12850.013,Y -481.830,Z 139.924,A 89.15631,B 0.00000,C 180.00000} ; retreat
  ; Step 2526, bar 2966
  LIN {X -12850.013,Y -481.830,Z 1050.408,A 90.84369,B 0.00000,C 180.00000} ; outside
  LIN {X -12850.013,Y -481.830,Z 89.924,A 90.84369,B 0.00000,C 180.00000} ; preinsert
  LIN {X -12850.013,Y -481.830,Z -160.076,A 90.84369,B 0.00000,C 180.00000} ; insert
  LIN {X -12850.013,Y -481.830,Z -160.076,A 90.84369,B 0.00000,C 180.00000} ; release
  LIN {X -12850.013,Y -481.830,Z 139.924,A 90.84369,B 0.00000,C 180.00000} ; retreat
  ; Step 2527, bar 2946
  LIN {X -12850.013,Y 481.830,Z 1050.408,A -90.84369,B 0.00000,C -180.00000} ; outside
  LIN {X -12850.013,Y 481.830,Z 89.924,A -90.84369,B 0.00000,C -180.00000} ; preinsert
  LIN {X -12850.013,Y 481.830,Z -160.076,A -90.84369,B 0.00000,C -180.00000} ; insert
  LIN {X -12850.013,Y 481.830,Z -160.076,A -90.84369,B 0.00000,C -180.00000} ; release
  LIN {X -12850.013,Y 481.830,Z 139.924,A -90.84369,B 0.00000,C -180.00000} ; retreat
  ; Step 2528, bar 2985
  LIN {X 12850.013,Y 481.830,Z 1050.408,A -89.15631,B 0.00000,C -180.00000} ; outside
  LIN {X 12850.013,Y 481.830,Z 89.924,A -89.15631,B 0.00000,C -180.00000} ; preinsert
  LIN {X 12850.013,Y 481.830,Z -160.076,A -89.15631,B 0.00000,C -180.00000} ; insert
  LIN {X 12850.013,Y 481.830,Z -160.076,A -89.15631,B 0.00000,C -180.00000} ; release
  LIN {X 12850.013,Y 481.830,Z 139.924,A -89.15631,B 0.00000,C -180.00000} ; retreat
  ; Step 2529, bar 272
  LIN {X -16249.715,Y 0.490,Z 1162.532,A 89.89089,B 0.00000,C 180.00000} ; outside
  LIN {X -16249.715,Y 0.490,Z 205.355,A 89.89089,B 0.00000,C 180.00000} ; preinsert
  LIN {X -16249.715,Y 0.490,Z -44.645,A 89.89089,B 0.00000,C 180.00000} ; insert
  LIN {X -16249.715,Y 0.490,Z -44.645,A 89.89089,B 0.00000,C 180.00000} ; release
  LIN {X -16249.715,Y 0.490,Z 255.355,A 89.89089,B 0.00000,C 180.00000} ; retreat
  ; Step 2530, bar 271
  LIN {X -16149.715,Y 0.490,Z 1162.532,A 89.89089,B 0.00000,C 180.00000} ; outside
  LIN {X -16149.715,Y 0.490,Z 205.355,A 89.89089,B 0.00000,C 180.00000} ; preinsert
  LIN {X -16149.715,Y 0.490,Z -44.645,A 89.89089,B 0.00000,C 180.00000} ; insert
  LIN {X -16149.715,Y 0.490,Z -44.645,A 89.89089,B 0.00000,C 180.00000} ; release
  LIN {X -16149.715,Y 0.490,Z 255.355,A 89.89089,B 0.00000,C 180.00000} ; retreat
  ; Step 2531, bar 270
  LIN {X -16049.715,Y 0.490,Z 1162.532,A 89.89089,B 0.00000,C 180.00000} ; outside
  LIN {X -16049.715,Y 0.490,Z 205.355,A 89.89089,B 0.00000,C 180.00000} ; preinsert
  LIN {X -16049.715,Y 0.490,Z -44.645,A 89.89089,B 0.00000,C 180.00000} ; insert
  LIN {X -16049.715,Y 0.490,Z -44.645,A 89.89089,B 0.00000,C 180.00000} ; release
  LIN {X -16049.715,Y 0.490,Z 255.355,A 89.89089,B 0.00000,C 180.00000} ; retreat
  ; Step 2532, bar 269
  LIN {X -15949.715,Y 0.490,Z 1162.532,A 89.89089,B 0.00000,C 180.00000} ; outside
  LIN {X -15949.715,Y 0.490,Z 205.355,A 89.89089,B 0.00000,C 180.00000} ; preinsert
  LIN {X -15949.715,Y 0.490,Z -44.645,A 89.89089,B 0.00000,C 180.00000} ; insert
  LIN {X -15949.715,Y 0.490,Z -44.645,A 89.89089,B 0.00000,C 180.00000} ; release
  LIN {X -15949.715,Y 0.490,Z 255.355,A 89.89089,B 0.00000,C 180.00000} ; retreat
  ; Step 2533, bar 268
  LIN {X -15849.715,Y 0.490,Z 1162.532,A 89.89089,B 0.00000,C 180.00000} ; outside
  LIN {X -15849.715,Y 0.490,Z 205.355,A 89.89089,B 0.00000,C 180.00000} ; preinsert
  LIN {X -15849.715,Y 0.490,Z -44.645,A 89.89089,B 0.00000,C 180.00000} ; insert
  LIN {X -15849.715,Y 0.490,Z -44.645,A 89.89089,B 0.00000,C 180.00000} ; release
  LIN {X -15849.715,Y 0.490,Z 255.355,A 89.89089,B 0.00000,C 180.00000} ; retreat
  ; Step 2534, bar 267
  LIN {X -15749.715,Y 0.490,Z 1162.532,A 89.89089,B 0.00000,C 180.00000} ; outside
  LIN {X -15749.715,Y 0.490,Z 205.355,A 89.89089,B 0.00000,C 180.00000} ; preinsert
  LIN {X -15749.715,Y 0.490,Z -44.645,A 89.89089,B 0.00000,C 180.00000} ; insert
  LIN {X -15749.715,Y 0.490,Z -44.645,A 89.89089,B 0.00000,C 180.00000} ; release
  LIN {X -15749.715,Y 0.490,Z 255.355,A 89.89089,B 0.00000,C 180.00000} ; retreat
  ; Step 2535, bar 266
  LIN {X -15649.715,Y 0.490,Z 1162.532,A 89.89089,B 0.00000,C 180.00000} ; outside
  LIN {X -15649.715,Y 0.490,Z 205.355,A 89.89089,B 0.00000,C 180.00000} ; preinsert
  LIN {X -15649.715,Y 0.490,Z -44.645,A 89.89089,B 0.00000,C 180.00000} ; insert
  LIN {X -15649.715,Y 0.490,Z -44.645,A 89.89089,B 0.00000,C 180.00000} ; release
  LIN {X -15649.715,Y 0.490,Z 255.355,A 89.89089,B 0.00000,C 180.00000} ; retreat
  ; Step 2536, bar 265
  LIN {X -15449.715,Y 0.490,Z 1162.532,A 89.89089,B 0.00000,C 180.00000} ; outside
  LIN {X -15449.715,Y 0.490,Z 205.355,A 89.89089,B 0.00000,C 180.00000} ; preinsert
  LIN {X -15449.715,Y 0.490,Z -44.645,A 89.89089,B 0.00000,C 180.00000} ; insert
  LIN {X -15449.715,Y 0.490,Z -44.645,A 89.89089,B 0.00000,C 180.00000} ; release
  LIN {X -15449.715,Y 0.490,Z 255.355,A 89.89089,B 0.00000,C 180.00000} ; retreat
  ; Step 2537, bar 264
  LIN {X -15349.715,Y 0.490,Z 1162.532,A 89.89089,B 0.00000,C 180.00000} ; outside
  LIN {X -15349.715,Y 0.490,Z 205.355,A 89.89089,B 0.00000,C 180.00000} ; preinsert
  LIN {X -15349.715,Y 0.490,Z -44.645,A 89.89089,B 0.00000,C 180.00000} ; insert
  LIN {X -15349.715,Y 0.490,Z -44.645,A 89.89089,B 0.00000,C 180.00000} ; release
  LIN {X -15349.715,Y 0.490,Z 255.355,A 89.89089,B 0.00000,C 180.00000} ; retreat
  ; Step 2538, bar 263
  LIN {X -15249.715,Y 0.490,Z 1162.532,A 89.89089,B 0.00000,C 180.00000} ; outside
  LIN {X -15249.715,Y 0.490,Z 205.355,A 89.89089,B 0.00000,C 180.00000} ; preinsert
  LIN {X -15249.715,Y 0.490,Z -44.645,A 89.89089,B 0.00000,C 180.00000} ; insert
  LIN {X -15249.715,Y 0.490,Z -44.645,A 89.89089,B 0.00000,C 180.00000} ; release
  LIN {X -15249.715,Y 0.490,Z 255.355,A 89.89089,B 0.00000,C 180.00000} ; retreat
  ; Step 2539, bar 262
  LIN {X -15149.715,Y 0.490,Z 1162.532,A 89.89089,B 0.00000,C 180.00000} ; outside
  LIN {X -15149.715,Y 0.490,Z 205.355,A 89.89089,B 0.00000,C 180.00000} ; preinsert
  LIN {X -15149.715,Y 0.490,Z -44.645,A 89.89089,B 0.00000,C 180.00000} ; insert
  LIN {X -15149.715,Y 0.490,Z -44.645,A 89.89089,B 0.00000,C 180.00000} ; release
  LIN {X -15149.715,Y 0.490,Z 255.355,A 89.89089,B 0.00000,C 180.00000} ; retreat
  ; Step 2540, bar 261
  LIN {X -15049.715,Y 0.490,Z 1162.532,A 89.89089,B 0.00000,C 180.00000} ; outside
  LIN {X -15049.715,Y 0.490,Z 205.355,A 89.89089,B 0.00000,C 180.00000} ; preinsert
  LIN {X -15049.715,Y 0.490,Z -44.645,A 89.89089,B 0.00000,C 180.00000} ; insert
  LIN {X -15049.715,Y 0.490,Z -44.645,A 89.89089,B 0.00000,C 180.00000} ; release
  LIN {X -15049.715,Y 0.490,Z 255.355,A 89.89089,B 0.00000,C 180.00000} ; retreat
  ; Step 2541, bar 260
  LIN {X -14949.715,Y 0.490,Z 1162.532,A 89.89089,B 0.00000,C 180.00000} ; outside
  LIN {X -14949.715,Y 0.490,Z 205.355,A 89.89089,B 0.00000,C 180.00000} ; preinsert
  LIN {X -14949.715,Y 0.490,Z -44.645,A 89.89089,B 0.00000,C 180.00000} ; insert
  LIN {X -14949.715,Y 0.490,Z -44.645,A 89.89089,B 0.00000,C 180.00000} ; release
  LIN {X -14949.715,Y 0.490,Z 255.355,A 89.89089,B 0.00000,C 180.00000} ; retreat
  ; Step 2542, bar 259
  LIN {X -14849.715,Y 0.490,Z 1162.532,A 89.89089,B 0.00000,C 180.00000} ; outside
  LIN {X -14849.715,Y 0.490,Z 205.355,A 89.89089,B 0.00000,C 180.00000} ; preinsert
  LIN {X -14849.715,Y 0.490,Z -44.645,A 89.89089,B 0.00000,C 180.00000} ; insert
  LIN {X -14849.715,Y 0.490,Z -44.645,A 89.89089,B 0.00000,C 180.00000} ; release
  LIN {X -14849.715,Y 0.490,Z 255.355,A 89.89089,B 0.00000,C 180.00000} ; retreat
  ; Step 2543, bar 258
  LIN {X -14749.715,Y 0.490,Z 1162.532,A 89.89089,B 0.00000,C 180.00000} ; outside
  LIN {X -14749.715,Y 0.490,Z 205.355,A 89.89089,B 0.00000,C 180.00000} ; preinsert
  LIN {X -14749.715,Y 0.490,Z -44.645,A 89.89089,B 0.00000,C 180.00000} ; insert
  LIN {X -14749.715,Y 0.490,Z -44.645,A 89.89089,B 0.00000,C 180.00000} ; release
  LIN {X -14749.715,Y 0.490,Z 255.355,A 89.89089,B 0.00000,C 180.00000} ; retreat
  ; Step 2544, bar 257
  LIN {X -14649.715,Y 0.490,Z 1162.532,A 89.89089,B 0.00000,C 180.00000} ; outside
  LIN {X -14649.715,Y 0.490,Z 205.355,A 89.89089,B 0.00000,C 180.00000} ; preinsert
  LIN {X -14649.715,Y 0.490,Z -44.645,A 89.89089,B 0.00000,C 180.00000} ; insert
  LIN {X -14649.715,Y 0.490,Z -44.645,A 89.89089,B 0.00000,C 180.00000} ; release
  LIN {X -14649.715,Y 0.490,Z 255.355,A 89.89089,B 0.00000,C 180.00000} ; retreat
  ; Step 2545, bar 256
  LIN {X -14449.715,Y 0.490,Z 1162.532,A 89.89089,B 0.00000,C 180.00000} ; outside
  LIN {X -14449.715,Y 0.490,Z 205.355,A 89.89089,B 0.00000,C 180.00000} ; preinsert
  LIN {X -14449.715,Y 0.490,Z -44.645,A 89.89089,B 0.00000,C 180.00000} ; insert
  LIN {X -14449.715,Y 0.490,Z -44.645,A 89.89089,B 0.00000,C 180.00000} ; release
  LIN {X -14449.715,Y 0.490,Z 255.355,A 89.89089,B 0.00000,C 180.00000} ; retreat
  ; Step 2546, bar 255
  LIN {X -14349.715,Y 0.490,Z 1162.532,A 89.89089,B 0.00000,C 180.00000} ; outside
  LIN {X -14349.715,Y 0.490,Z 205.355,A 89.89089,B 0.00000,C 180.00000} ; preinsert
  LIN {X -14349.715,Y 0.490,Z -44.645,A 89.89089,B 0.00000,C 180.00000} ; insert
  LIN {X -14349.715,Y 0.490,Z -44.645,A 89.89089,B 0.00000,C 180.00000} ; release
  LIN {X -14349.715,Y 0.490,Z 255.355,A 89.89089,B 0.00000,C 180.00000} ; retreat
  ; Step 2547, bar 254
  LIN {X -14249.715,Y 0.490,Z 1162.532,A 89.89089,B 0.00000,C 180.00000} ; outside
  LIN {X -14249.715,Y 0.490,Z 205.355,A 89.89089,B 0.00000,C 180.00000} ; preinsert
  LIN {X -14249.715,Y 0.490,Z -44.645,A 89.89089,B 0.00000,C 180.00000} ; insert
  LIN {X -14249.715,Y 0.490,Z -44.645,A 89.89089,B 0.00000,C 180.00000} ; release
  LIN {X -14249.715,Y 0.490,Z 255.355,A 89.89089,B 0.00000,C 180.00000} ; retreat
  ; Step 2548, bar 253
  LIN {X -14149.715,Y 0.490,Z 1162.532,A 89.89089,B 0.00000,C 180.00000} ; outside
  LIN {X -14149.715,Y 0.490,Z 205.355,A 89.89089,B 0.00000,C 180.00000} ; preinsert
  LIN {X -14149.715,Y 0.490,Z -44.645,A 89.89089,B 0.00000,C 180.00000} ; insert
  LIN {X -14149.715,Y 0.490,Z -44.645,A 89.89089,B 0.00000,C 180.00000} ; release
  LIN {X -14149.715,Y 0.490,Z 255.355,A 89.89089,B 0.00000,C 180.00000} ; retreat
  ; Step 2549, bar 252
  LIN {X -13849.715,Y 0.490,Z 1162.532,A 89.89089,B 0.00000,C 180.00000} ; outside
  LIN {X -13849.715,Y 0.490,Z 205.355,A 89.89089,B 0.00000,C 180.00000} ; preinsert
  LIN {X -13849.715,Y 0.490,Z -44.645,A 89.89089,B 0.00000,C 180.00000} ; insert
  LIN {X -13849.715,Y 0.490,Z -44.645,A 89.89089,B 0.00000,C 180.00000} ; release
  LIN {X -13849.715,Y 0.490,Z 255.355,A 89.89089,B 0.00000,C 180.00000} ; retreat
  ; Step 2550, bar 251
  LIN {X -13749.715,Y 0.490,Z 1162.532,A 89.89089,B 0.00000,C 180.00000} ; outside
  LIN {X -13749.715,Y 0.490,Z 205.355,A 89.89089,B 0.00000,C 180.00000} ; preinsert
  LIN {X -13749.715,Y 0.490,Z -44.645,A 89.89089,B 0.00000,C 180.00000} ; insert
  LIN {X -13749.715,Y 0.490,Z -44.645,A 89.89089,B 0.00000,C 180.00000} ; release
  LIN {X -13749.715,Y 0.490,Z 255.355,A 89.89089,B 0.00000,C 180.00000} ; retreat
  ; Step 2551, bar 113
  LIN {X 13749.715,Y 0.490,Z 1162.532,A 90.10911,B 0.00000,C 180.00000} ; outside
  LIN {X 13749.715,Y 0.490,Z 205.355,A 90.10911,B 0.00000,C 180.00000} ; preinsert
  LIN {X 13749.715,Y 0.490,Z -44.645,A 90.10911,B 0.00000,C 180.00000} ; insert
  LIN {X 13749.715,Y 0.490,Z -44.645,A 90.10911,B 0.00000,C 180.00000} ; release
  LIN {X 13749.715,Y 0.490,Z 255.355,A 90.10911,B 0.00000,C 180.00000} ; retreat
  ; Step 2552, bar 114
  LIN {X 13849.715,Y 0.490,Z 1162.532,A 90.10911,B 0.00000,C 180.00000} ; outside
  LIN {X 13849.715,Y 0.490,Z 205.355,A 90.10911,B 0.00000,C 180.00000} ; preinsert
  LIN {X 13849.715,Y 0.490,Z -44.645,A 90.10911,B 0.00000,C 180.00000} ; insert
  LIN {X 13849.715,Y 0.490,Z -44.645,A 90.10911,B 0.00000,C 180.00000} ; release
  LIN {X 13849.715,Y 0.490,Z 255.355,A 90.10911,B 0.00000,C 180.00000} ; retreat
  ; Step 2553, bar 117
  LIN {X 14149.715,Y 0.490,Z 1162.532,A 90.10911,B 0.00000,C 180.00000} ; outside
  LIN {X 14149.715,Y 0.490,Z 205.355,A 90.10911,B 0.00000,C 180.00000} ; preinsert
  LIN {X 14149.715,Y 0.490,Z -44.645,A 90.10911,B 0.00000,C 180.00000} ; insert
  LIN {X 14149.715,Y 0.490,Z -44.645,A 90.10911,B 0.00000,C 180.00000} ; release
  LIN {X 14149.715,Y 0.490,Z 255.355,A 90.10911,B 0.00000,C 180.00000} ; retreat
  ; Step 2554, bar 118
  LIN {X 14249.715,Y 0.490,Z 1162.532,A 90.10911,B 0.00000,C 180.00000} ; outside
  LIN {X 14249.715,Y 0.490,Z 205.355,A 90.10911,B 0.00000,C 180.00000} ; preinsert
  LIN {X 14249.715,Y 0.490,Z -44.645,A 90.10911,B 0.00000,C 180.00000} ; insert
  LIN {X 14249.715,Y 0.490,Z -44.645,A 90.10911,B 0.00000,C 180.00000} ; release
  LIN {X 14249.715,Y 0.490,Z 255.355,A 90.10911,B 0.00000,C 180.00000} ; retreat
  ; Step 2555, bar 119
  LIN {X 14349.715,Y 0.490,Z 1162.532,A 90.10911,B 0.00000,C 180.00000} ; outside
  LIN {X 14349.715,Y 0.490,Z 205.355,A 90.10911,B 0.00000,C 180.00000} ; preinsert
  LIN {X 14349.715,Y 0.490,Z -44.645,A 90.10911,B 0.00000,C 180.00000} ; insert
  LIN {X 14349.715,Y 0.490,Z -44.645,A 90.10911,B 0.00000,C 180.00000} ; release
  LIN {X 14349.715,Y 0.490,Z 255.355,A 90.10911,B 0.00000,C 180.00000} ; retreat
  ; Step 2556, bar 120
  LIN {X 14449.715,Y 0.490,Z 1162.532,A 90.10911,B 0.00000,C 180.00000} ; outside
  LIN {X 14449.715,Y 0.490,Z 205.355,A 90.10911,B 0.00000,C 180.00000} ; preinsert
  LIN {X 14449.715,Y 0.490,Z -44.645,A 90.10911,B 0.00000,C 180.00000} ; insert
  LIN {X 14449.715,Y 0.490,Z -44.645,A 90.10911,B 0.00000,C 180.00000} ; release
  LIN {X 14449.715,Y 0.490,Z 255.355,A 90.10911,B 0.00000,C 180.00000} ; retreat
  ; Step 2557, bar 122
  LIN {X 14649.715,Y 0.490,Z 1162.532,A 90.10911,B 0.00000,C 180.00000} ; outside
  LIN {X 14649.715,Y 0.490,Z 205.355,A 90.10911,B 0.00000,C 180.00000} ; preinsert
  LIN {X 14649.715,Y 0.490,Z -44.645,A 90.10911,B 0.00000,C 180.00000} ; insert
  LIN {X 14649.715,Y 0.490,Z -44.645,A 90.10911,B 0.00000,C 180.00000} ; release
  LIN {X 14649.715,Y 0.490,Z 255.355,A 90.10911,B 0.00000,C 180.00000} ; retreat
  ; Step 2558, bar 123
  LIN {X 14749.715,Y 0.490,Z 1162.532,A 90.10911,B 0.00000,C 180.00000} ; outside
  LIN {X 14749.715,Y 0.490,Z 205.355,A 90.10911,B 0.00000,C 180.00000} ; preinsert
  LIN {X 14749.715,Y 0.490,Z -44.645,A 90.10911,B 0.00000,C 180.00000} ; insert
  LIN {X 14749.715,Y 0.490,Z -44.645,A 90.10911,B 0.00000,C 180.00000} ; release
  LIN {X 14749.715,Y 0.490,Z 255.355,A 90.10911,B 0.00000,C 180.00000} ; retreat
  ; Step 2559, bar 124
  LIN {X 14849.715,Y 0.490,Z 1162.532,A 90.10911,B 0.00000,C 180.00000} ; outside
  LIN {X 14849.715,Y 0.490,Z 205.355,A 90.10911,B 0.00000,C 180.00000} ; preinsert
  LIN {X 14849.715,Y 0.490,Z -44.645,A 90.10911,B 0.00000,C 180.00000} ; insert
  LIN {X 14849.715,Y 0.490,Z -44.645,A 90.10911,B 0.00000,C 180.00000} ; release
  LIN {X 14849.715,Y 0.490,Z 255.355,A 90.10911,B 0.00000,C 180.00000} ; retreat
  ; Step 2560, bar 125
  LIN {X 14949.715,Y 0.490,Z 1162.532,A 90.10911,B 0.00000,C 180.00000} ; outside
  LIN {X 14949.715,Y 0.490,Z 205.355,A 90.10911,B 0.00000,C 180.00000} ; preinsert
  LIN {X 14949.715,Y 0.490,Z -44.645,A 90.10911,B 0.00000,C 180.00000} ; insert
  LIN {X 14949.715,Y 0.490,Z -44.645,A 90.10911,B 0.00000,C 180.00000} ; release
  LIN {X 14949.715,Y 0.490,Z 255.355,A 90.10911,B 0.00000,C 180.00000} ; retreat
  ; Step 2561, bar 126
  LIN {X 15049.715,Y 0.490,Z 1162.532,A 90.10911,B 0.00000,C 180.00000} ; outside
  LIN {X 15049.715,Y 0.490,Z 205.355,A 90.10911,B 0.00000,C 180.00000} ; preinsert
  LIN {X 15049.715,Y 0.490,Z -44.645,A 90.10911,B 0.00000,C 180.00000} ; insert
  LIN {X 15049.715,Y 0.490,Z -44.645,A 90.10911,B 0.00000,C 180.00000} ; release
  LIN {X 15049.715,Y 0.490,Z 255.355,A 90.10911,B 0.00000,C 180.00000} ; retreat
  ; Step 2562, bar 127
  LIN {X 15149.715,Y 0.490,Z 1162.532,A 90.10911,B 0.00000,C 180.00000} ; outside
  LIN {X 15149.715,Y 0.490,Z 205.355,A 90.10911,B 0.00000,C 180.00000} ; preinsert
  LIN {X 15149.715,Y 0.490,Z -44.645,A 90.10911,B 0.00000,C 180.00000} ; insert
  LIN {X 15149.715,Y 0.490,Z -44.645,A 90.10911,B 0.00000,C 180.00000} ; release
  LIN {X 15149.715,Y 0.490,Z 255.355,A 90.10911,B 0.00000,C 180.00000} ; retreat
  ; Step 2563, bar 128
  LIN {X 15249.715,Y 0.490,Z 1162.532,A 90.10911,B 0.00000,C 180.00000} ; outside
  LIN {X 15249.715,Y 0.490,Z 205.355,A 90.10911,B 0.00000,C 180.00000} ; preinsert
  LIN {X 15249.715,Y 0.490,Z -44.645,A 90.10911,B 0.00000,C 180.00000} ; insert
  LIN {X 15249.715,Y 0.490,Z -44.645,A 90.10911,B 0.00000,C 180.00000} ; release
  LIN {X 15249.715,Y 0.490,Z 255.355,A 90.10911,B 0.00000,C 180.00000} ; retreat
  ; Step 2564, bar 129
  LIN {X 15349.715,Y 0.490,Z 1162.532,A 90.10911,B 0.00000,C 180.00000} ; outside
  LIN {X 15349.715,Y 0.490,Z 205.355,A 90.10911,B 0.00000,C 180.00000} ; preinsert
  LIN {X 15349.715,Y 0.490,Z -44.645,A 90.10911,B 0.00000,C 180.00000} ; insert
  LIN {X 15349.715,Y 0.490,Z -44.645,A 90.10911,B 0.00000,C 180.00000} ; release
  LIN {X 15349.715,Y 0.490,Z 255.355,A 90.10911,B 0.00000,C 180.00000} ; retreat
  ; Step 2565, bar 130
  LIN {X 15449.715,Y 0.490,Z 1162.532,A 90.10911,B 0.00000,C 180.00000} ; outside
  LIN {X 15449.715,Y 0.490,Z 205.355,A 90.10911,B 0.00000,C 180.00000} ; preinsert
  LIN {X 15449.715,Y 0.490,Z -44.645,A 90.10911,B 0.00000,C 180.00000} ; insert
  LIN {X 15449.715,Y 0.490,Z -44.645,A 90.10911,B 0.00000,C 180.00000} ; release
  LIN {X 15449.715,Y 0.490,Z 255.355,A 90.10911,B 0.00000,C 180.00000} ; retreat
  ; Step 2566, bar 132
  LIN {X 15649.715,Y 0.490,Z 1162.532,A 90.10911,B 0.00000,C 180.00000} ; outside
  LIN {X 15649.715,Y 0.490,Z 205.355,A 90.10911,B 0.00000,C 180.00000} ; preinsert
  LIN {X 15649.715,Y 0.490,Z -44.645,A 90.10911,B 0.00000,C 180.00000} ; insert
  LIN {X 15649.715,Y 0.490,Z -44.645,A 90.10911,B 0.00000,C 180.00000} ; release
  LIN {X 15649.715,Y 0.490,Z 255.355,A 90.10911,B 0.00000,C 180.00000} ; retreat
  ; Step 2567, bar 133
  LIN {X 15749.715,Y 0.490,Z 1162.532,A 90.10911,B 0.00000,C 180.00000} ; outside
  LIN {X 15749.715,Y 0.490,Z 205.355,A 90.10911,B 0.00000,C 180.00000} ; preinsert
  LIN {X 15749.715,Y 0.490,Z -44.645,A 90.10911,B 0.00000,C 180.00000} ; insert
  LIN {X 15749.715,Y 0.490,Z -44.645,A 90.10911,B 0.00000,C 180.00000} ; release
  LIN {X 15749.715,Y 0.490,Z 255.355,A 90.10911,B 0.00000,C 180.00000} ; retreat
  ; Step 2568, bar 134
  LIN {X 15849.715,Y 0.490,Z 1162.532,A 90.10911,B 0.00000,C 180.00000} ; outside
  LIN {X 15849.715,Y 0.490,Z 205.355,A 90.10911,B 0.00000,C 180.00000} ; preinsert
  LIN {X 15849.715,Y 0.490,Z -44.645,A 90.10911,B 0.00000,C 180.00000} ; insert
  LIN {X 15849.715,Y 0.490,Z -44.645,A 90.10911,B 0.00000,C 180.00000} ; release
  LIN {X 15849.715,Y 0.490,Z 255.355,A 90.10911,B 0.00000,C 180.00000} ; retreat
  ; Step 2569, bar 135
  LIN {X 15949.715,Y 0.490,Z 1162.532,A 90.10911,B 0.00000,C 180.00000} ; outside
  LIN {X 15949.715,Y 0.490,Z 205.355,A 90.10911,B 0.00000,C 180.00000} ; preinsert
  LIN {X 15949.715,Y 0.490,Z -44.645,A 90.10911,B 0.00000,C 180.00000} ; insert
  LIN {X 15949.715,Y 0.490,Z -44.645,A 90.10911,B 0.00000,C 180.00000} ; release
  LIN {X 15949.715,Y 0.490,Z 255.355,A 90.10911,B 0.00000,C 180.00000} ; retreat
  ; Step 2570, bar 136
  LIN {X 16049.715,Y 0.490,Z 1162.532,A 90.10911,B 0.00000,C 180.00000} ; outside
  LIN {X 16049.715,Y 0.490,Z 205.355,A 90.10911,B 0.00000,C 180.00000} ; preinsert
  LIN {X 16049.715,Y 0.490,Z -44.645,A 90.10911,B 0.00000,C 180.00000} ; insert
  LIN {X 16049.715,Y 0.490,Z -44.645,A 90.10911,B 0.00000,C 180.00000} ; release
  LIN {X 16049.715,Y 0.490,Z 255.355,A 90.10911,B 0.00000,C 180.00000} ; retreat
  ; Step 2571, bar 137
  LIN {X 16149.715,Y 0.490,Z 1162.532,A 90.10911,B 0.00000,C 180.00000} ; outside
  LIN {X 16149.715,Y 0.490,Z 205.355,A 90.10911,B 0.00000,C 180.00000} ; preinsert
  LIN {X 16149.715,Y 0.490,Z -44.645,A 90.10911,B 0.00000,C 180.00000} ; insert
  LIN {X 16149.715,Y 0.490,Z -44.645,A 90.10911,B 0.00000,C 180.00000} ; release
  LIN {X 16149.715,Y 0.490,Z 255.355,A 90.10911,B 0.00000,C 180.00000} ; retreat
  ; Step 2572, bar 138
  LIN {X 16249.715,Y 0.490,Z 1162.532,A 90.10911,B 0.00000,C 180.00000} ; outside
  LIN {X 16249.715,Y 0.490,Z 205.355,A 90.10911,B 0.00000,C 180.00000} ; preinsert
  LIN {X 16249.715,Y 0.490,Z -44.645,A 90.10911,B 0.00000,C 180.00000} ; insert
  LIN {X 16249.715,Y 0.490,Z -44.645,A 90.10911,B 0.00000,C 180.00000} ; release
  LIN {X 16249.715,Y 0.490,Z 255.355,A 90.10911,B 0.00000,C 180.00000} ; retreat
  ; Step 2573, bar 15
  LIN {X 2000.043,Y 0.301,Z 1164.708,A 89.93710,B 0.00000,C 180.00000} ; outside
  LIN {X 2000.043,Y 0.301,Z 206.219,A 89.93710,B 0.00000,C 180.00000} ; preinsert
  LIN {X 2000.043,Y 0.301,Z -43.781,A 89.93710,B 0.00000,C 180.00000} ; insert
  LIN {X 2000.043,Y 0.301,Z -43.781,A 89.93710,B 0.00000,C 180.00000} ; release
  LIN {X 2000.043,Y 0.301,Z 256.219,A 89.93710,B 0.00000,C 180.00000} ; retreat
  ; Step 2574, bar 47
  LIN {X 6000.043,Y 0.301,Z 1164.708,A 89.93710,B 0.00000,C 180.00000} ; outside
  LIN {X 6000.043,Y 0.301,Z 206.219,A 89.93710,B 0.00000,C 180.00000} ; preinsert
  LIN {X 6000.043,Y 0.301,Z -43.781,A 89.93710,B 0.00000,C 180.00000} ; insert
  LIN {X 6000.043,Y 0.301,Z -43.781,A 89.93710,B 0.00000,C 180.00000} ; release
  LIN {X 6000.043,Y 0.301,Z 256.219,A 89.93710,B 0.00000,C 180.00000} ; retreat
  ; Step 2575, bar 79
  LIN {X 10000.043,Y 0.301,Z 1164.708,A 89.93710,B 0.00000,C 180.00000} ; outside
  LIN {X 10000.043,Y 0.301,Z 206.219,A 89.93710,B 0.00000,C 180.00000} ; preinsert
  LIN {X 10000.043,Y 0.301,Z -43.781,A 89.93710,B 0.00000,C 180.00000} ; insert
  LIN {X 10000.043,Y 0.301,Z -43.781,A 89.93710,B 0.00000,C 180.00000} ; release
  LIN {X 10000.043,Y 0.301,Z 256.219,A 89.93710,B 0.00000,C 180.00000} ; retreat
  ; Step 2576, bar 250
  LIN {X -10000.043,Y 0.302,Z 1164.708,A 90.06290,B 0.00000,C 180.00000} ; outside
  LIN {X -10000.043,Y 0.302,Z 206.219,A 90.06290,B 0.00000,C 180.00000} ; preinsert
  LIN {X -10000.043,Y 0.302,Z -43.781,A 90.06290,B 0.00000,C 180.00000} ; insert
  LIN {X -10000.043,Y 0.302,Z -43.781,A 90.06290,B 0.00000,C 180.00000} ; release
  LIN {X -10000.043,Y 0.302,Z 256.219,A 90.06290,B 0.00000,C 180.00000} ; retreat
  ; Step 2577, bar 249
  LIN {X -6000.043,Y 0.302,Z 1164.708,A 90.06290,B 0.00000,C 180.00000} ; outside
  LIN {X -6000.043,Y 0.302,Z 206.219,A 90.06290,B 0.00000,C 180.00000} ; preinsert
  LIN {X -6000.043,Y 0.302,Z -43.781,A 90.06290,B 0.00000,C 180.00000} ; insert
  LIN {X -6000.043,Y 0.302,Z -43.781,A 90.06290,B 0.00000,C 180.00000} ; release
  LIN {X -6000.043,Y 0.302,Z 256.219,A 90.06290,B 0.00000,C 180.00000} ; retreat
  ; Step 2578, bar 248
  LIN {X -2000.043,Y 0.302,Z 1164.708,A 90.06290,B 0.00000,C 180.00000} ; outside
  LIN {X -2000.043,Y 0.302,Z 206.219,A 90.06290,B 0.00000,C 180.00000} ; preinsert
  LIN {X -2000.043,Y 0.302,Z -43.781,A 90.06290,B 0.00000,C 180.00000} ; insert
  LIN {X -2000.043,Y 0.302,Z -43.781,A 90.06290,B 0.00000,C 180.00000} ; release
  LIN {X -2000.043,Y 0.302,Z 256.219,A 90.06290,B 0.00000,C 180.00000} ; retreat
  ; Step 2579, bar 276
  LIN {X -15550.467,Y 0.150,Z 1163.461,A -89.91334,B 0.00000,C 180.00000} ; outside
  LIN {X -15550.467,Y 0.150,Z 205.930,A -89.91334,B 0.00000,C 180.00000} ; preinsert
  LIN {X -15550.467,Y 0.150,Z -44.070,A -89.91334,B 0.00000,C 180.00000} ; insert
  LIN {X -15550.467,Y 0.150,Z -44.070,A -89.91334,B 0.00000,C 180.00000} ; release
  LIN {X -15550.467,Y 0.150,Z 255.930,A -89.91334,B 0.00000,C 180.00000} ; retreat
  ; Step 2580, bar 275
  LIN {X -14550.467,Y 0.150,Z 1163.461,A -89.91334,B 0.00000,C 180.00000} ; outside
  LIN {X -14550.467,Y 0.150,Z 205.930,A -89.91334,B 0.00000,C 180.00000} ; preinsert
  LIN {X -14550.467,Y 0.150,Z -44.070,A -89.91334,B 0.00000,C 180.00000} ; insert
  LIN {X -14550.467,Y 0.150,Z -44.070,A -89.91334,B 0.00000,C 180.00000} ; release
  LIN {X -14550.467,Y 0.150,Z 255.930,A -89.91334,B 0.00000,C 180.00000} ; retreat
  ; Step 2581, bar 247
  LIN {X -13649.998,Y -0.298,Z 1164.733,A -90.00011,B 0.00000,C -180.00000} ; outside
  LIN {X -13649.998,Y -0.298,Z 206.498,A -90.00011,B 0.00000,C -180.00000} ; preinsert
  LIN {X -13649.998,Y -0.298,Z -43.502,A -90.00011,B 0.00000,C -180.00000} ; insert
  LIN {X -13649.998,Y -0.298,Z -43.502,A -90.00011,B 0.00000,C -180.00000} ; release
  LIN {X -13649.998,Y -0.298,Z 256.498,A -90.00011,B 0.00000,C -180.00000} ; retreat
  ; Step 2582, bar 246
  LIN {X -13549.998,Y -0.298,Z 1164.733,A -90.00011,B 0.00000,C -180.00000} ; outside
  LIN {X -13549.998,Y -0.298,Z 206.498,A -90.00011,B 0.00000,C -180.00000} ; preinsert
  LIN {X -13549.998,Y -0.298,Z -43.502,A -90.00011,B 0.00000,C -180.00000} ; insert
  LIN {X -13549.998,Y -0.298,Z -43.502,A -90.00011,B 0.00000,C -180.00000} ; release
  LIN {X -13549.998,Y -0.298,Z 256.498,A -90.00011,B 0.00000,C -180.00000} ; retreat
  ; Step 2583, bar 245
  LIN {X -13449.998,Y -0.298,Z 1164.733,A -90.00011,B 0.00000,C -180.00000} ; outside
  LIN {X -13449.998,Y -0.298,Z 206.498,A -90.00011,B 0.00000,C -180.00000} ; preinsert
  LIN {X -13449.998,Y -0.298,Z -43.502,A -90.00011,B 0.00000,C -180.00000} ; insert
  LIN {X -13449.998,Y -0.298,Z -43.502,A -90.00011,B 0.00000,C -180.00000} ; release
  LIN {X -13449.998,Y -0.298,Z 256.498,A -90.00011,B 0.00000,C -180.00000} ; retreat
  ; Step 2584, bar 244
  LIN {X -13349.998,Y -0.298,Z 1164.733,A -90.00011,B 0.00000,C -180.00000} ; outside
  LIN {X -13349.998,Y -0.298,Z 206.498,A -90.00011,B 0.00000,C -180.00000} ; preinsert
  LIN {X -13349.998,Y -0.298,Z -43.502,A -90.00011,B 0.00000,C -180.00000} ; insert
  LIN {X -13349.998,Y -0.298,Z -43.502,A -90.00011,B 0.00000,C -180.00000} ; release
  LIN {X -13349.998,Y -0.298,Z 256.498,A -90.00011,B 0.00000,C -180.00000} ; retreat
  ; Step 2585, bar 243
  LIN {X -13249.998,Y -0.298,Z 1164.733,A -90.00011,B 0.00000,C -180.00000} ; outside
  LIN {X -13249.998,Y -0.298,Z 206.498,A -90.00011,B 0.00000,C -180.00000} ; preinsert
  LIN {X -13249.998,Y -0.298,Z -43.502,A -90.00011,B 0.00000,C -180.00000} ; insert
  LIN {X -13249.998,Y -0.298,Z -43.502,A -90.00011,B 0.00000,C -180.00000} ; release
  LIN {X -13249.998,Y -0.298,Z 256.498,A -90.00011,B 0.00000,C -180.00000} ; retreat
  ; Step 2586, bar 242
  LIN {X -13149.998,Y -0.298,Z 1164.733,A -90.00011,B 0.00000,C -180.00000} ; outside
  LIN {X -13149.998,Y -0.298,Z 206.498,A -90.00011,B 0.00000,C -180.00000} ; preinsert
  LIN {X -13149.998,Y -0.298,Z -43.502,A -90.00011,B 0.00000,C -180.00000} ; insert
  LIN {X -13149.998,Y -0.298,Z -43.502,A -90.00011,B 0.00000,C -180.00000} ; release
  LIN {X -13149.998,Y -0.298,Z 256.498,A -90.00011,B 0.00000,C -180.00000} ; retreat
  ; Step 2587, bar 241
  LIN {X -13049.998,Y -0.298,Z 1164.733,A -90.00011,B 0.00000,C -180.00000} ; outside
  LIN {X -13049.998,Y -0.298,Z 206.498,A -90.00011,B 0.00000,C -180.00000} ; preinsert
  LIN {X -13049.998,Y -0.298,Z -43.502,A -90.00011,B 0.00000,C -180.00000} ; insert
  LIN {X -13049.998,Y -0.298,Z -43.502,A -90.00011,B 0.00000,C -180.00000} ; release
  LIN {X -13049.998,Y -0.298,Z 256.498,A -90.00011,B 0.00000,C -180.00000} ; retreat
  ; Step 2588, bar 240
  LIN {X -12949.998,Y -0.298,Z 1164.733,A -90.00011,B 0.00000,C -180.00000} ; outside
  LIN {X -12949.998,Y -0.298,Z 206.498,A -90.00011,B 0.00000,C -180.00000} ; preinsert
  LIN {X -12949.998,Y -0.298,Z -43.502,A -90.00011,B 0.00000,C -180.00000} ; insert
  LIN {X -12949.998,Y -0.298,Z -43.502,A -90.00011,B 0.00000,C -180.00000} ; release
  LIN {X -12949.998,Y -0.298,Z 256.498,A -90.00011,B 0.00000,C -180.00000} ; retreat
  ; Step 2589, bar 239
  LIN {X -12849.998,Y -0.298,Z 1164.733,A -90.00011,B 0.00000,C -180.00000} ; outside
  LIN {X -12849.998,Y -0.298,Z 206.498,A -90.00011,B 0.00000,C -180.00000} ; preinsert
  LIN {X -12849.998,Y -0.298,Z -43.502,A -90.00011,B 0.00000,C -180.00000} ; insert
  LIN {X -12849.998,Y -0.298,Z -43.502,A -90.00011,B 0.00000,C -180.00000} ; release
  LIN {X -12849.998,Y -0.298,Z 256.498,A -90.00011,B 0.00000,C -180.00000} ; retreat
  ; Step 2590, bar 238
  LIN {X -12749.998,Y -0.298,Z 1164.733,A -90.00011,B 0.00000,C -180.00000} ; outside
  LIN {X -12749.998,Y -0.298,Z 206.498,A -90.00011,B 0.00000,C -180.00000} ; preinsert
  LIN {X -12749.998,Y -0.298,Z -43.502,A -90.00011,B 0.00000,C -180.00000} ; insert
  LIN {X -12749.998,Y -0.298,Z -43.502,A -90.00011,B 0.00000,C -180.00000} ; release
  LIN {X -12749.998,Y -0.298,Z 256.498,A -90.00011,B 0.00000,C -180.00000} ; retreat
  ; Step 2591, bar 237
  LIN {X -12649.998,Y -0.298,Z 1164.733,A -90.00011,B 0.00000,C -180.00000} ; outside
  LIN {X -12649.998,Y -0.298,Z 206.498,A -90.00011,B 0.00000,C -180.00000} ; preinsert
  LIN {X -12649.998,Y -0.298,Z -43.502,A -90.00011,B 0.00000,C -180.00000} ; insert
  LIN {X -12649.998,Y -0.298,Z -43.502,A -90.00011,B 0.00000,C -180.00000} ; release
  LIN {X -12649.998,Y -0.298,Z 256.498,A -90.00011,B 0.00000,C -180.00000} ; retreat
  ; Step 2592, bar 236
  LIN {X -12549.998,Y -0.298,Z 1164.733,A -90.00011,B 0.00000,C -180.00000} ; outside
  LIN {X -12549.998,Y -0.298,Z 206.498,A -90.00011,B 0.00000,C -180.00000} ; preinsert
  LIN {X -12549.998,Y -0.298,Z -43.502,A -90.00011,B 0.00000,C -180.00000} ; insert
  LIN {X -12549.998,Y -0.298,Z -43.502,A -90.00011,B 0.00000,C -180.00000} ; release
  LIN {X -12549.998,Y -0.298,Z 256.498,A -90.00011,B 0.00000,C -180.00000} ; retreat
  ; Step 2593, bar 235
  LIN {X -12449.998,Y -0.298,Z 1164.733,A -90.00011,B 0.00000,C -180.00000} ; outside
  LIN {X -12449.998,Y -0.298,Z 206.498,A -90.00011,B 0.00000,C -180.00000} ; preinsert
  LIN {X -12449.998,Y -0.298,Z -43.502,A -90.00011,B 0.00000,C -180.00000} ; insert
  LIN {X -12449.998,Y -0.298,Z -43.502,A -90.00011,B 0.00000,C -180.00000} ; release
  LIN {X -12449.998,Y -0.298,Z 256.498,A -90.00011,B 0.00000,C -180.00000} ; retreat
  ; Step 2594, bar 234
  LIN {X -12349.998,Y -0.298,Z 1164.733,A -90.00011,B 0.00000,C -180.00000} ; outside
  LIN {X -12349.998,Y -0.298,Z 206.498,A -90.00011,B 0.00000,C -180.00000} ; preinsert
  LIN {X -12349.998,Y -0.298,Z -43.502,A -90.00011,B 0.00000,C -180.00000} ; insert
  LIN {X -12349.998,Y -0.298,Z -43.502,A -90.00011,B 0.00000,C -180.00000} ; release
  LIN {X -12349.998,Y -0.298,Z 256.498,A -90.00011,B 0.00000,C -180.00000} ; retreat
  ; Step 2595, bar 233
  LIN {X -12249.998,Y -0.298,Z 1164.733,A -90.00011,B 0.00000,C -180.00000} ; outside
  LIN {X -12249.998,Y -0.298,Z 206.498,A -90.00011,B 0.00000,C -180.00000} ; preinsert
  LIN {X -12249.998,Y -0.298,Z -43.502,A -90.00011,B 0.00000,C -180.00000} ; insert
  LIN {X -12249.998,Y -0.298,Z -43.502,A -90.00011,B 0.00000,C -180.00000} ; release
  LIN {X -12249.998,Y -0.298,Z 256.498,A -90.00011,B 0.00000,C -180.00000} ; retreat
  ; Step 2596, bar 232
  LIN {X -12124.998,Y -0.298,Z 1164.733,A -90.00011,B 0.00000,C -180.00000} ; outside
  LIN {X -12124.998,Y -0.298,Z 206.498,A -90.00011,B 0.00000,C -180.00000} ; preinsert
  LIN {X -12124.998,Y -0.298,Z -43.502,A -90.00011,B 0.00000,C -180.00000} ; insert
  LIN {X -12124.998,Y -0.298,Z -43.502,A -90.00011,B 0.00000,C -180.00000} ; release
  LIN {X -12124.998,Y -0.298,Z 256.498,A -90.00011,B 0.00000,C -180.00000} ; retreat
  ; Step 2597, bar 231
  LIN {X -11999.998,Y -0.298,Z 1164.733,A -90.00011,B 0.00000,C -180.00000} ; outside
  LIN {X -11999.998,Y -0.298,Z 206.498,A -90.00011,B 0.00000,C -180.00000} ; preinsert
  LIN {X -11999.998,Y -0.298,Z -43.502,A -90.00011,B 0.00000,C -180.00000} ; insert
  LIN {X -11999.998,Y -0.298,Z -43.502,A -90.00011,B 0.00000,C -180.00000} ; release
  LIN {X -11999.998,Y -0.298,Z 256.498,A -90.00011,B 0.00000,C -180.00000} ; retreat
  ; Step 2598, bar 230
  LIN {X -11874.998,Y -0.298,Z 1164.733,A -90.00011,B 0.00000,C -180.00000} ; outside
  LIN {X -11874.998,Y -0.298,Z 206.498,A -90.00011,B 0.00000,C -180.00000} ; preinsert
  LIN {X -11874.998,Y -0.298,Z -43.502,A -90.00011,B 0.00000,C -180.00000} ; insert
  LIN {X -11874.998,Y -0.298,Z -43.502,A -90.00011,B 0.00000,C -180.00000} ; release
  LIN {X -11874.998,Y -0.298,Z 256.498,A -90.00011,B 0.00000,C -180.00000} ; retreat
  ; Step 2599, bar 229
  LIN {X -11749.998,Y -0.298,Z 1164.733,A -90.00011,B 0.00000,C -180.00000} ; outside
  LIN {X -11749.998,Y -0.298,Z 206.498,A -90.00011,B 0.00000,C -180.00000} ; preinsert
  LIN {X -11749.998,Y -0.298,Z -43.502,A -90.00011,B 0.00000,C -180.00000} ; insert
  LIN {X -11749.998,Y -0.298,Z -43.502,A -90.00011,B 0.00000,C -180.00000} ; release
  LIN {X -11749.998,Y -0.298,Z 256.498,A -90.00011,B 0.00000,C -180.00000} ; retreat
  ; Step 2600, bar 228
  LIN {X -11624.998,Y -0.298,Z 1164.733,A -90.00011,B 0.00000,C -180.00000} ; outside
  LIN {X -11624.998,Y -0.298,Z 206.498,A -90.00011,B 0.00000,C -180.00000} ; preinsert
  LIN {X -11624.998,Y -0.298,Z -43.502,A -90.00011,B 0.00000,C -180.00000} ; insert
  LIN {X -11624.998,Y -0.298,Z -43.502,A -90.00011,B 0.00000,C -180.00000} ; release
  LIN {X -11624.998,Y -0.298,Z 256.498,A -90.00011,B 0.00000,C -180.00000} ; retreat
  ; Step 2601, bar 227
  LIN {X -11499.998,Y -0.298,Z 1164.733,A -90.00011,B 0.00000,C -180.00000} ; outside
  LIN {X -11499.998,Y -0.298,Z 206.498,A -90.00011,B 0.00000,C -180.00000} ; preinsert
  LIN {X -11499.998,Y -0.298,Z -43.502,A -90.00011,B 0.00000,C -180.00000} ; insert
  LIN {X -11499.998,Y -0.298,Z -43.502,A -90.00011,B 0.00000,C -180.00000} ; release
  LIN {X -11499.998,Y -0.298,Z 256.498,A -90.00011,B 0.00000,C -180.00000} ; retreat
  ; Step 2602, bar 226
  LIN {X -11374.998,Y -0.298,Z 1164.733,A -90.00011,B 0.00000,C -180.00000} ; outside
  LIN {X -11374.998,Y -0.298,Z 206.498,A -90.00011,B 0.00000,C -180.00000} ; preinsert
  LIN {X -11374.998,Y -0.298,Z -43.502,A -90.00011,B 0.00000,C -180.00000} ; insert
  LIN {X -11374.998,Y -0.298,Z -43.502,A -90.00011,B 0.00000,C -180.00000} ; release
  LIN {X -11374.998,Y -0.298,Z 256.498,A -90.00011,B 0.00000,C -180.00000} ; retreat
  ; Step 2603, bar 225
  LIN {X -11249.998,Y -0.298,Z 1164.733,A -90.00011,B 0.00000,C -180.00000} ; outside
  LIN {X -11249.998,Y -0.298,Z 206.498,A -90.00011,B 0.00000,C -180.00000} ; preinsert
  LIN {X -11249.998,Y -0.298,Z -43.502,A -90.00011,B 0.00000,C -180.00000} ; insert
  LIN {X -11249.998,Y -0.298,Z -43.502,A -90.00011,B 0.00000,C -180.00000} ; release
  LIN {X -11249.998,Y -0.298,Z 256.498,A -90.00011,B 0.00000,C -180.00000} ; retreat
  ; Step 2604, bar 224
  LIN {X -11124.998,Y -0.298,Z 1164.733,A -90.00011,B 0.00000,C -180.00000} ; outside
  LIN {X -11124.998,Y -0.298,Z 206.498,A -90.00011,B 0.00000,C -180.00000} ; preinsert
  LIN {X -11124.998,Y -0.298,Z -43.502,A -90.00011,B 0.00000,C -180.00000} ; insert
  LIN {X -11124.998,Y -0.298,Z -43.502,A -90.00011,B 0.00000,C -180.00000} ; release
  LIN {X -11124.998,Y -0.298,Z 256.498,A -90.00011,B 0.00000,C -180.00000} ; retreat
  ; Step 2605, bar 223
  LIN {X -10999.998,Y -0.298,Z 1164.733,A -90.00011,B 0.00000,C -180.00000} ; outside
  LIN {X -10999.998,Y -0.298,Z 206.498,A -90.00011,B 0.00000,C -180.00000} ; preinsert
  LIN {X -10999.998,Y -0.298,Z -43.502,A -90.00011,B 0.00000,C -180.00000} ; insert
  LIN {X -10999.998,Y -0.298,Z -43.502,A -90.00011,B 0.00000,C -180.00000} ; release
  LIN {X -10999.998,Y -0.298,Z 256.498,A -90.00011,B 0.00000,C -180.00000} ; retreat
  ; Step 2606, bar 222
  LIN {X -10874.998,Y -0.298,Z 1164.733,A -90.00011,B 0.00000,C -180.00000} ; outside
  LIN {X -10874.998,Y -0.298,Z 206.498,A -90.00011,B 0.00000,C -180.00000} ; preinsert
  LIN {X -10874.998,Y -0.298,Z -43.502,A -90.00011,B 0.00000,C -180.00000} ; insert
  LIN {X -10874.998,Y -0.298,Z -43.502,A -90.00011,B 0.00000,C -180.00000} ; release
  LIN {X -10874.998,Y -0.298,Z 256.498,A -90.00011,B 0.00000,C -180.00000} ; retreat
  ; Step 2607, bar 221
  LIN {X -10749.998,Y -0.298,Z 1164.733,A -90.00011,B 0.00000,C -180.00000} ; outside
  LIN {X -10749.998,Y -0.298,Z 206.498,A -90.00011,B 0.00000,C -180.00000} ; preinsert
  LIN {X -10749.998,Y -0.298,Z -43.502,A -90.00011,B 0.00000,C -180.00000} ; insert
  LIN {X -10749.998,Y -0.298,Z -43.502,A -90.00011,B 0.00000,C -180.00000} ; release
  LIN {X -10749.998,Y -0.298,Z 256.498,A -90.00011,B 0.00000,C -180.00000} ; retreat
  ; Step 2608, bar 220
  LIN {X -10624.998,Y -0.298,Z 1164.733,A -90.00011,B 0.00000,C -180.00000} ; outside
  LIN {X -10624.998,Y -0.298,Z 206.498,A -90.00011,B 0.00000,C -180.00000} ; preinsert
  LIN {X -10624.998,Y -0.298,Z -43.502,A -90.00011,B 0.00000,C -180.00000} ; insert
  LIN {X -10624.998,Y -0.298,Z -43.502,A -90.00011,B 0.00000,C -180.00000} ; release
  LIN {X -10624.998,Y -0.298,Z 256.498,A -90.00011,B 0.00000,C -180.00000} ; retreat
  ; Step 2609, bar 219
  LIN {X -10499.998,Y -0.298,Z 1164.733,A -90.00011,B 0.00000,C -180.00000} ; outside
  LIN {X -10499.998,Y -0.298,Z 206.498,A -90.00011,B 0.00000,C -180.00000} ; preinsert
  LIN {X -10499.998,Y -0.298,Z -43.502,A -90.00011,B 0.00000,C -180.00000} ; insert
  LIN {X -10499.998,Y -0.298,Z -43.502,A -90.00011,B 0.00000,C -180.00000} ; release
  LIN {X -10499.998,Y -0.298,Z 256.498,A -90.00011,B 0.00000,C -180.00000} ; retreat
  ; Step 2610, bar 218
  LIN {X -10374.998,Y -0.298,Z 1164.733,A -90.00011,B 0.00000,C -180.00000} ; outside
  LIN {X -10374.998,Y -0.298,Z 206.498,A -90.00011,B 0.00000,C -180.00000} ; preinsert
  LIN {X -10374.998,Y -0.298,Z -43.502,A -90.00011,B 0.00000,C -180.00000} ; insert
  LIN {X -10374.998,Y -0.298,Z -43.502,A -90.00011,B 0.00000,C -180.00000} ; release
  LIN {X -10374.998,Y -0.298,Z 256.498,A -90.00011,B 0.00000,C -180.00000} ; retreat
  ; Step 2611, bar 217
  LIN {X -10249.998,Y -0.298,Z 1164.733,A -90.00011,B 0.00000,C -180.00000} ; outside
  LIN {X -10249.998,Y -0.298,Z 206.498,A -90.00011,B 0.00000,C -180.00000} ; preinsert
  LIN {X -10249.998,Y -0.298,Z -43.502,A -90.00011,B 0.00000,C -180.00000} ; insert
  LIN {X -10249.998,Y -0.298,Z -43.502,A -90.00011,B 0.00000,C -180.00000} ; release
  LIN {X -10249.998,Y -0.298,Z 256.498,A -90.00011,B 0.00000,C -180.00000} ; retreat
  ; Step 2612, bar 216
  LIN {X -10124.998,Y -0.298,Z 1164.733,A -90.00011,B 0.00000,C -180.00000} ; outside
  LIN {X -10124.998,Y -0.298,Z 206.498,A -90.00011,B 0.00000,C -180.00000} ; preinsert
  LIN {X -10124.998,Y -0.298,Z -43.502,A -90.00011,B 0.00000,C -180.00000} ; insert
  LIN {X -10124.998,Y -0.298,Z -43.502,A -90.00011,B 0.00000,C -180.00000} ; release
  LIN {X -10124.998,Y -0.298,Z 256.498,A -90.00011,B 0.00000,C -180.00000} ; retreat
  ; Step 2613, bar 215
  LIN {X -9874.998,Y -0.298,Z 1164.733,A -90.00011,B 0.00000,C -180.00000} ; outside
  LIN {X -9874.998,Y -0.298,Z 206.498,A -90.00011,B 0.00000,C -180.00000} ; preinsert
  LIN {X -9874.998,Y -0.298,Z -43.502,A -90.00011,B 0.00000,C -180.00000} ; insert
  LIN {X -9874.998,Y -0.298,Z -43.502,A -90.00011,B 0.00000,C -180.00000} ; release
  LIN {X -9874.998,Y -0.298,Z 256.498,A -90.00011,B 0.00000,C -180.00000} ; retreat
  ; Step 2614, bar 214
  LIN {X -9749.998,Y -0.298,Z 1164.733,A -90.00011,B 0.00000,C -180.00000} ; outside
  LIN {X -9749.998,Y -0.298,Z 206.498,A -90.00011,B 0.00000,C -180.00000} ; preinsert
  LIN {X -9749.998,Y -0.298,Z -43.502,A -90.00011,B 0.00000,C -180.00000} ; insert
  LIN {X -9749.998,Y -0.298,Z -43.502,A -90.00011,B 0.00000,C -180.00000} ; release
  LIN {X -9749.998,Y -0.298,Z 256.498,A -90.00011,B 0.00000,C -180.00000} ; retreat
  ; Step 2615, bar 213
  LIN {X -9624.998,Y -0.298,Z 1164.733,A -90.00011,B 0.00000,C -180.00000} ; outside
  LIN {X -9624.998,Y -0.298,Z 206.498,A -90.00011,B 0.00000,C -180.00000} ; preinsert
  LIN {X -9624.998,Y -0.298,Z -43.502,A -90.00011,B 0.00000,C -180.00000} ; insert
  LIN {X -9624.998,Y -0.298,Z -43.502,A -90.00011,B 0.00000,C -180.00000} ; release
  LIN {X -9624.998,Y -0.298,Z 256.498,A -90.00011,B 0.00000,C -180.00000} ; retreat
  ; Step 2616, bar 212
  LIN {X -9499.998,Y -0.298,Z 1164.733,A -90.00011,B 0.00000,C -180.00000} ; outside
  LIN {X -9499.998,Y -0.298,Z 206.498,A -90.00011,B 0.00000,C -180.00000} ; preinsert
  LIN {X -9499.998,Y -0.298,Z -43.502,A -90.00011,B 0.00000,C -180.00000} ; insert
  LIN {X -9499.998,Y -0.298,Z -43.502,A -90.00011,B 0.00000,C -180.00000} ; release
  LIN {X -9499.998,Y -0.298,Z 256.498,A -90.00011,B 0.00000,C -180.00000} ; retreat
  ; Step 2617, bar 211
  LIN {X -9374.998,Y -0.298,Z 1164.733,A -90.00011,B 0.00000,C -180.00000} ; outside
  LIN {X -9374.998,Y -0.298,Z 206.498,A -90.00011,B 0.00000,C -180.00000} ; preinsert
  LIN {X -9374.998,Y -0.298,Z -43.502,A -90.00011,B 0.00000,C -180.00000} ; insert
  LIN {X -9374.998,Y -0.298,Z -43.502,A -90.00011,B 0.00000,C -180.00000} ; release
  LIN {X -9374.998,Y -0.298,Z 256.498,A -90.00011,B 0.00000,C -180.00000} ; retreat
  ; Step 2618, bar 210
  LIN {X -9249.998,Y -0.298,Z 1164.733,A -90.00011,B 0.00000,C -180.00000} ; outside
  LIN {X -9249.998,Y -0.298,Z 206.498,A -90.00011,B 0.00000,C -180.00000} ; preinsert
  LIN {X -9249.998,Y -0.298,Z -43.502,A -90.00011,B 0.00000,C -180.00000} ; insert
  LIN {X -9249.998,Y -0.298,Z -43.502,A -90.00011,B 0.00000,C -180.00000} ; release
  LIN {X -9249.998,Y -0.298,Z 256.498,A -90.00011,B 0.00000,C -180.00000} ; retreat
  ; Step 2619, bar 209
  LIN {X -9124.998,Y -0.298,Z 1164.733,A -90.00011,B 0.00000,C -180.00000} ; outside
  LIN {X -9124.998,Y -0.298,Z 206.498,A -90.00011,B 0.00000,C -180.00000} ; preinsert
  LIN {X -9124.998,Y -0.298,Z -43.502,A -90.00011,B 0.00000,C -180.00000} ; insert
  LIN {X -9124.998,Y -0.298,Z -43.502,A -90.00011,B 0.00000,C -180.00000} ; release
  LIN {X -9124.998,Y -0.298,Z 256.498,A -90.00011,B 0.00000,C -180.00000} ; retreat
  ; Step 2620, bar 208
  LIN {X -8999.998,Y -0.298,Z 1164.733,A -90.00011,B 0.00000,C -180.00000} ; outside
  LIN {X -8999.998,Y -0.298,Z 206.498,A -90.00011,B 0.00000,C -180.00000} ; preinsert
  LIN {X -8999.998,Y -0.298,Z -43.502,A -90.00011,B 0.00000,C -180.00000} ; insert
  LIN {X -8999.998,Y -0.298,Z -43.502,A -90.00011,B 0.00000,C -180.00000} ; release
  LIN {X -8999.998,Y -0.298,Z 256.498,A -90.00011,B 0.00000,C -180.00000} ; retreat
  ; Step 2621, bar 207
  LIN {X -8874.998,Y -0.298,Z 1164.733,A -90.00011,B 0.00000,C -180.00000} ; outside
  LIN {X -8874.998,Y -0.298,Z 206.498,A -90.00011,B 0.00000,C -180.00000} ; preinsert
  LIN {X -8874.998,Y -0.298,Z -43.502,A -90.00011,B 0.00000,C -180.00000} ; insert
  LIN {X -8874.998,Y -0.298,Z -43.502,A -90.00011,B 0.00000,C -180.00000} ; release
  LIN {X -8874.998,Y -0.298,Z 256.498,A -90.00011,B 0.00000,C -180.00000} ; retreat
  ; Step 2622, bar 206
  LIN {X -8749.998,Y -0.298,Z 1164.733,A -90.00011,B 0.00000,C -180.00000} ; outside
  LIN {X -8749.998,Y -0.298,Z 206.498,A -90.00011,B 0.00000,C -180.00000} ; preinsert
  LIN {X -8749.998,Y -0.298,Z -43.502,A -90.00011,B 0.00000,C -180.00000} ; insert
  LIN {X -8749.998,Y -0.298,Z -43.502,A -90.00011,B 0.00000,C -180.00000} ; release
  LIN {X -8749.998,Y -0.298,Z 256.498,A -90.00011,B 0.00000,C -180.00000} ; retreat
  ; Step 2623, bar 205
  LIN {X -8624.998,Y -0.298,Z 1164.733,A -90.00011,B 0.00000,C -180.00000} ; outside
  LIN {X -8624.998,Y -0.298,Z 206.498,A -90.00011,B 0.00000,C -180.00000} ; preinsert
  LIN {X -8624.998,Y -0.298,Z -43.502,A -90.00011,B 0.00000,C -180.00000} ; insert
  LIN {X -8624.998,Y -0.298,Z -43.502,A -90.00011,B 0.00000,C -180.00000} ; release
  LIN {X -8624.998,Y -0.298,Z 256.498,A -90.00011,B 0.00000,C -180.00000} ; retreat
  ; Step 2624, bar 204
  LIN {X -8499.998,Y -0.298,Z 1164.733,A -90.00011,B 0.00000,C -180.00000} ; outside
  LIN {X -8499.998,Y -0.298,Z 206.498,A -90.00011,B 0.00000,C -180.00000} ; preinsert
  LIN {X -8499.998,Y -0.298,Z -43.502,A -90.00011,B 0.00000,C -180.00000} ; insert
  LIN {X -8499.998,Y -0.298,Z -43.502,A -90.00011,B 0.00000,C -180.00000} ; release
  LIN {X -8499.998,Y -0.298,Z 256.498,A -90.00011,B 0.00000,C -180.00000} ; retreat
  ; Step 2625, bar 203
  LIN {X -8374.998,Y -0.298,Z 1164.733,A -90.00011,B 0.00000,C -180.00000} ; outside
  LIN {X -8374.998,Y -0.298,Z 206.498,A -90.00011,B 0.00000,C -180.00000} ; preinsert
  LIN {X -8374.998,Y -0.298,Z -43.502,A -90.00011,B 0.00000,C -180.00000} ; insert
  LIN {X -8374.998,Y -0.298,Z -43.502,A -90.00011,B 0.00000,C -180.00000} ; release
  LIN {X -8374.998,Y -0.298,Z 256.498,A -90.00011,B 0.00000,C -180.00000} ; retreat
  ; Step 2626, bar 202
  LIN {X -8249.998,Y -0.298,Z 1164.733,A -90.00011,B 0.00000,C -180.00000} ; outside
  LIN {X -8249.998,Y -0.298,Z 206.498,A -90.00011,B 0.00000,C -180.00000} ; preinsert
  LIN {X -8249.998,Y -0.298,Z -43.502,A -90.00011,B 0.00000,C -180.00000} ; insert
  LIN {X -8249.998,Y -0.298,Z -43.502,A -90.00011,B 0.00000,C -180.00000} ; release
  LIN {X -8249.998,Y -0.298,Z 256.498,A -90.00011,B 0.00000,C -180.00000} ; retreat
  ; Step 2627, bar 201
  LIN {X -8124.998,Y -0.298,Z 1164.733,A -90.00011,B 0.00000,C -180.00000} ; outside
  LIN {X -8124.998,Y -0.298,Z 206.498,A -90.00011,B 0.00000,C -180.00000} ; preinsert
  LIN {X -8124.998,Y -0.298,Z -43.502,A -90.00011,B 0.00000,C -180.00000} ; insert
  LIN {X -8124.998,Y -0.298,Z -43.502,A -90.00011,B 0.00000,C -180.00000} ; release
  LIN {X -8124.998,Y -0.298,Z 256.498,A -90.00011,B 0.00000,C -180.00000} ; retreat
  ; Step 2628, bar 200
  LIN {X -7999.998,Y -0.298,Z 1164.733,A -90.00011,B 0.00000,C -180.00000} ; outside
  LIN {X -7999.998,Y -0.298,Z 206.498,A -90.00011,B 0.00000,C -180.00000} ; preinsert
  LIN {X -7999.998,Y -0.298,Z -43.502,A -90.00011,B 0.00000,C -180.00000} ; insert
  LIN {X -7999.998,Y -0.298,Z -43.502,A -90.00011,B 0.00000,C -180.00000} ; release
  LIN {X -7999.998,Y -0.298,Z 256.498,A -90.00011,B 0.00000,C -180.00000} ; retreat
  ; Step 2629, bar 199
  LIN {X -7874.998,Y -0.298,Z 1164.733,A -90.00011,B 0.00000,C -180.00000} ; outside
  LIN {X -7874.998,Y -0.298,Z 206.498,A -90.00011,B 0.00000,C -180.00000} ; preinsert
  LIN {X -7874.998,Y -0.298,Z -43.502,A -90.00011,B 0.00000,C -180.00000} ; insert
  LIN {X -7874.998,Y -0.298,Z -43.502,A -90.00011,B 0.00000,C -180.00000} ; release
  LIN {X -7874.998,Y -0.298,Z 256.498,A -90.00011,B 0.00000,C -180.00000} ; retreat
  ; Step 2630, bar 198
  LIN {X -7749.998,Y -0.298,Z 1164.733,A -90.00011,B 0.00000,C -180.00000} ; outside
  LIN {X -7749.998,Y -0.298,Z 206.498,A -90.00011,B 0.00000,C -180.00000} ; preinsert
  LIN {X -7749.998,Y -0.298,Z -43.502,A -90.00011,B 0.00000,C -180.00000} ; insert
  LIN {X -7749.998,Y -0.298,Z -43.502,A -90.00011,B 0.00000,C -180.00000} ; release
  LIN {X -7749.998,Y -0.298,Z 256.498,A -90.00011,B 0.00000,C -180.00000} ; retreat
  ; Step 2631, bar 197
  LIN {X -7624.998,Y -0.298,Z 1164.733,A -90.00011,B 0.00000,C -180.00000} ; outside
  LIN {X -7624.998,Y -0.298,Z 206.498,A -90.00011,B 0.00000,C -180.00000} ; preinsert
  LIN {X -7624.998,Y -0.298,Z -43.502,A -90.00011,B 0.00000,C -180.00000} ; insert
  LIN {X -7624.998,Y -0.298,Z -43.502,A -90.00011,B 0.00000,C -180.00000} ; release
  LIN {X -7624.998,Y -0.298,Z 256.498,A -90.00011,B 0.00000,C -180.00000} ; retreat
  ; Step 2632, bar 196
  LIN {X -7499.998,Y -0.298,Z 1164.733,A -90.00011,B 0.00000,C -180.00000} ; outside
  LIN {X -7499.998,Y -0.298,Z 206.498,A -90.00011,B 0.00000,C -180.00000} ; preinsert
  LIN {X -7499.998,Y -0.298,Z -43.502,A -90.00011,B 0.00000,C -180.00000} ; insert
  LIN {X -7499.998,Y -0.298,Z -43.502,A -90.00011,B 0.00000,C -180.00000} ; release
  LIN {X -7499.998,Y -0.298,Z 256.498,A -90.00011,B 0.00000,C -180.00000} ; retreat
  ; Step 2633, bar 195
  LIN {X -7374.998,Y -0.298,Z 1164.733,A -90.00011,B 0.00000,C -180.00000} ; outside
  LIN {X -7374.998,Y -0.298,Z 206.498,A -90.00011,B 0.00000,C -180.00000} ; preinsert
  LIN {X -7374.998,Y -0.298,Z -43.502,A -90.00011,B 0.00000,C -180.00000} ; insert
  LIN {X -7374.998,Y -0.298,Z -43.502,A -90.00011,B 0.00000,C -180.00000} ; release
  LIN {X -7374.998,Y -0.298,Z 256.498,A -90.00011,B 0.00000,C -180.00000} ; retreat
  ; Step 2634, bar 194
  LIN {X -7249.998,Y -0.298,Z 1164.733,A -90.00011,B 0.00000,C -180.00000} ; outside
  LIN {X -7249.998,Y -0.298,Z 206.498,A -90.00011,B 0.00000,C -180.00000} ; preinsert
  LIN {X -7249.998,Y -0.298,Z -43.502,A -90.00011,B 0.00000,C -180.00000} ; insert
  LIN {X -7249.998,Y -0.298,Z -43.502,A -90.00011,B 0.00000,C -180.00000} ; release
  LIN {X -7249.998,Y -0.298,Z 256.498,A -90.00011,B 0.00000,C -180.00000} ; retreat
  ; Step 2635, bar 193
  LIN {X -7124.998,Y -0.298,Z 1164.733,A -90.00011,B 0.00000,C -180.00000} ; outside
  LIN {X -7124.998,Y -0.298,Z 206.498,A -90.00011,B 0.00000,C -180.00000} ; preinsert
  LIN {X -7124.998,Y -0.298,Z -43.502,A -90.00011,B 0.00000,C -180.00000} ; insert
  LIN {X -7124.998,Y -0.298,Z -43.502,A -90.00011,B 0.00000,C -180.00000} ; release
  LIN {X -7124.998,Y -0.298,Z 256.498,A -90.00011,B 0.00000,C -180.00000} ; retreat
  ; Step 2636, bar 192
  LIN {X -6999.998,Y -0.298,Z 1164.733,A -90.00011,B 0.00000,C -180.00000} ; outside
  LIN {X -6999.998,Y -0.298,Z 206.498,A -90.00011,B 0.00000,C -180.00000} ; preinsert
  LIN {X -6999.998,Y -0.298,Z -43.502,A -90.00011,B 0.00000,C -180.00000} ; insert
  LIN {X -6999.998,Y -0.298,Z -43.502,A -90.00011,B 0.00000,C -180.00000} ; release
  LIN {X -6999.998,Y -0.298,Z 256.498,A -90.00011,B 0.00000,C -180.00000} ; retreat
  ; Step 2637, bar 191
  LIN {X -6874.998,Y -0.298,Z 1164.733,A -90.00011,B 0.00000,C -180.00000} ; outside
  LIN {X -6874.998,Y -0.298,Z 206.498,A -90.00011,B 0.00000,C -180.00000} ; preinsert
  LIN {X -6874.998,Y -0.298,Z -43.502,A -90.00011,B 0.00000,C -180.00000} ; insert
  LIN {X -6874.998,Y -0.298,Z -43.502,A -90.00011,B 0.00000,C -180.00000} ; release
  LIN {X -6874.998,Y -0.298,Z 256.498,A -90.00011,B 0.00000,C -180.00000} ; retreat
  ; Step 2638, bar 190
  LIN {X -6749.998,Y -0.298,Z 1164.733,A -90.00011,B 0.00000,C -180.00000} ; outside
  LIN {X -6749.998,Y -0.298,Z 206.498,A -90.00011,B 0.00000,C -180.00000} ; preinsert
  LIN {X -6749.998,Y -0.298,Z -43.502,A -90.00011,B 0.00000,C -180.00000} ; insert
  LIN {X -6749.998,Y -0.298,Z -43.502,A -90.00011,B 0.00000,C -180.00000} ; release
  LIN {X -6749.998,Y -0.298,Z 256.498,A -90.00011,B 0.00000,C -180.00000} ; retreat
  ; Step 2639, bar 189
  LIN {X -6624.998,Y -0.298,Z 1164.733,A -90.00011,B 0.00000,C -180.00000} ; outside
  LIN {X -6624.998,Y -0.298,Z 206.498,A -90.00011,B 0.00000,C -180.00000} ; preinsert
  LIN {X -6624.998,Y -0.298,Z -43.502,A -90.00011,B 0.00000,C -180.00000} ; insert
  LIN {X -6624.998,Y -0.298,Z -43.502,A -90.00011,B 0.00000,C -180.00000} ; release
  LIN {X -6624.998,Y -0.298,Z 256.498,A -90.00011,B 0.00000,C -180.00000} ; retreat
  ; Step 2640, bar 188
  LIN {X -6499.998,Y -0.298,Z 1164.733,A -90.00011,B 0.00000,C -180.00000} ; outside
  LIN {X -6499.998,Y -0.298,Z 206.498,A -90.00011,B 0.00000,C -180.00000} ; preinsert
  LIN {X -6499.998,Y -0.298,Z -43.502,A -90.00011,B 0.00000,C -180.00000} ; insert
  LIN {X -6499.998,Y -0.298,Z -43.502,A -90.00011,B 0.00000,C -180.00000} ; release
  LIN {X -6499.998,Y -0.298,Z 256.498,A -90.00011,B 0.00000,C -180.00000} ; retreat
  ; Step 2641, bar 187
  LIN {X -6374.998,Y -0.298,Z 1164.733,A -90.00011,B 0.00000,C -180.00000} ; outside
  LIN {X -6374.998,Y -0.298,Z 206.498,A -90.00011,B 0.00000,C -180.00000} ; preinsert
  LIN {X -6374.998,Y -0.298,Z -43.502,A -90.00011,B 0.00000,C -180.00000} ; insert
  LIN {X -6374.998,Y -0.298,Z -43.502,A -90.00011,B 0.00000,C -180.00000} ; release
  LIN {X -6374.998,Y -0.298,Z 256.498,A -90.00011,B 0.00000,C -180.00000} ; retreat
  ; Step 2642, bar 186
  LIN {X -6249.998,Y -0.298,Z 1164.733,A -90.00011,B 0.00000,C -180.00000} ; outside
  LIN {X -6249.998,Y -0.298,Z 206.498,A -90.00011,B 0.00000,C -180.00000} ; preinsert
  LIN {X -6249.998,Y -0.298,Z -43.502,A -90.00011,B 0.00000,C -180.00000} ; insert
  LIN {X -6249.998,Y -0.298,Z -43.502,A -90.00011,B 0.00000,C -180.00000} ; release
  LIN {X -6249.998,Y -0.298,Z 256.498,A -90.00011,B 0.00000,C -180.00000} ; retreat
  ; Step 2643, bar 185
  LIN {X -6124.998,Y -0.298,Z 1164.733,A -90.00011,B 0.00000,C -180.00000} ; outside
  LIN {X -6124.998,Y -0.298,Z 206.498,A -90.00011,B 0.00000,C -180.00000} ; preinsert
  LIN {X -6124.998,Y -0.298,Z -43.502,A -90.00011,B 0.00000,C -180.00000} ; insert
  LIN {X -6124.998,Y -0.298,Z -43.502,A -90.00011,B 0.00000,C -180.00000} ; release
  LIN {X -6124.998,Y -0.298,Z 256.498,A -90.00011,B 0.00000,C -180.00000} ; retreat
  ; Step 2644, bar 184
  LIN {X -5874.998,Y -0.298,Z 1164.733,A -90.00011,B 0.00000,C -180.00000} ; outside
  LIN {X -5874.998,Y -0.298,Z 206.498,A -90.00011,B 0.00000,C -180.00000} ; preinsert
  LIN {X -5874.998,Y -0.298,Z -43.502,A -90.00011,B 0.00000,C -180.00000} ; insert
  LIN {X -5874.998,Y -0.298,Z -43.502,A -90.00011,B 0.00000,C -180.00000} ; release
  LIN {X -5874.998,Y -0.298,Z 256.498,A -90.00011,B 0.00000,C -180.00000} ; retreat
  ; Step 2645, bar 183
  LIN {X -5749.998,Y -0.298,Z 1164.733,A -90.00011,B 0.00000,C -180.00000} ; outside
  LIN {X -5749.998,Y -0.298,Z 206.498,A -90.00011,B 0.00000,C -180.00000} ; preinsert
  LIN {X -5749.998,Y -0.298,Z -43.502,A -90.00011,B 0.00000,C -180.00000} ; insert
  LIN {X -5749.998,Y -0.298,Z -43.502,A -90.00011,B 0.00000,C -180.00000} ; release
  LIN {X -5749.998,Y -0.298,Z 256.498,A -90.00011,B 0.00000,C -180.00000} ; retreat
  ; Step 2646, bar 182
  LIN {X -5624.998,Y -0.298,Z 1164.733,A -90.00011,B 0.00000,C -180.00000} ; outside
  LIN {X -5624.998,Y -0.298,Z 206.498,A -90.00011,B 0.00000,C -180.00000} ; preinsert
  LIN {X -5624.998,Y -0.298,Z -43.502,A -90.00011,B 0.00000,C -180.00000} ; insert
  LIN {X -5624.998,Y -0.298,Z -43.502,A -90.00011,B 0.00000,C -180.00000} ; release
  LIN {X -5624.998,Y -0.298,Z 256.498,A -90.00011,B 0.00000,C -180.00000} ; retreat
  ; Step 2647, bar 181
  LIN {X -5499.998,Y -0.298,Z 1164.733,A -90.00011,B 0.00000,C -180.00000} ; outside
  LIN {X -5499.998,Y -0.298,Z 206.498,A -90.00011,B 0.00000,C -180.00000} ; preinsert
  LIN {X -5499.998,Y -0.298,Z -43.502,A -90.00011,B 0.00000,C -180.00000} ; insert
  LIN {X -5499.998,Y -0.298,Z -43.502,A -90.00011,B 0.00000,C -180.00000} ; release
  LIN {X -5499.998,Y -0.298,Z 256.498,A -90.00011,B 0.00000,C -180.00000} ; retreat
  ; Step 2648, bar 180
  LIN {X -5374.998,Y -0.298,Z 1164.733,A -90.00011,B 0.00000,C -180.00000} ; outside
  LIN {X -5374.998,Y -0.298,Z 206.498,A -90.00011,B 0.00000,C -180.00000} ; preinsert
  LIN {X -5374.998,Y -0.298,Z -43.502,A -90.00011,B 0.00000,C -180.00000} ; insert
  LIN {X -5374.998,Y -0.298,Z -43.502,A -90.00011,B 0.00000,C -180.00000} ; release
  LIN {X -5374.998,Y -0.298,Z 256.498,A -90.00011,B 0.00000,C -180.00000} ; retreat
  ; Step 2649, bar 179
  LIN {X -5249.998,Y -0.298,Z 1164.733,A -90.00011,B 0.00000,C -180.00000} ; outside
  LIN {X -5249.998,Y -0.298,Z 206.498,A -90.00011,B 0.00000,C -180.00000} ; preinsert
  LIN {X -5249.998,Y -0.298,Z -43.502,A -90.00011,B 0.00000,C -180.00000} ; insert
  LIN {X -5249.998,Y -0.298,Z -43.502,A -90.00011,B 0.00000,C -180.00000} ; release
  LIN {X -5249.998,Y -0.298,Z 256.498,A -90.00011,B 0.00000,C -180.00000} ; retreat
  ; Step 2650, bar 178
  LIN {X -5124.998,Y -0.298,Z 1164.733,A -90.00011,B 0.00000,C -180.00000} ; outside
  LIN {X -5124.998,Y -0.298,Z 206.498,A -90.00011,B 0.00000,C -180.00000} ; preinsert
  LIN {X -5124.998,Y -0.298,Z -43.502,A -90.00011,B 0.00000,C -180.00000} ; insert
  LIN {X -5124.998,Y -0.298,Z -43.502,A -90.00011,B 0.00000,C -180.00000} ; release
  LIN {X -5124.998,Y -0.298,Z 256.498,A -90.00011,B 0.00000,C -180.00000} ; retreat
  ; Step 2651, bar 177
  LIN {X -4999.998,Y -0.298,Z 1164.733,A -90.00011,B 0.00000,C -180.00000} ; outside
  LIN {X -4999.998,Y -0.298,Z 206.498,A -90.00011,B 0.00000,C -180.00000} ; preinsert
  LIN {X -4999.998,Y -0.298,Z -43.502,A -90.00011,B 0.00000,C -180.00000} ; insert
  LIN {X -4999.998,Y -0.298,Z -43.502,A -90.00011,B 0.00000,C -180.00000} ; release
  LIN {X -4999.998,Y -0.298,Z 256.498,A -90.00011,B 0.00000,C -180.00000} ; retreat
  ; Step 2652, bar 176
  LIN {X -4874.998,Y -0.298,Z 1164.733,A -90.00011,B 0.00000,C -180.00000} ; outside
  LIN {X -4874.998,Y -0.298,Z 206.498,A -90.00011,B 0.00000,C -180.00000} ; preinsert
  LIN {X -4874.998,Y -0.298,Z -43.502,A -90.00011,B 0.00000,C -180.00000} ; insert
  LIN {X -4874.998,Y -0.298,Z -43.502,A -90.00011,B 0.00000,C -180.00000} ; release
  LIN {X -4874.998,Y -0.298,Z 256.498,A -90.00011,B 0.00000,C -180.00000} ; retreat
  ; Step 2653, bar 175
  LIN {X -4749.998,Y -0.298,Z 1164.733,A -90.00011,B 0.00000,C -180.00000} ; outside
  LIN {X -4749.998,Y -0.298,Z 206.498,A -90.00011,B 0.00000,C -180.00000} ; preinsert
  LIN {X -4749.998,Y -0.298,Z -43.502,A -90.00011,B 0.00000,C -180.00000} ; insert
  LIN {X -4749.998,Y -0.298,Z -43.502,A -90.00011,B 0.00000,C -180.00000} ; release
  LIN {X -4749.998,Y -0.298,Z 256.498,A -90.00011,B 0.00000,C -180.00000} ; retreat
  ; Step 2654, bar 174
  LIN {X -4624.998,Y -0.298,Z 1164.733,A -90.00011,B 0.00000,C -180.00000} ; outside
  LIN {X -4624.998,Y -0.298,Z 206.498,A -90.00011,B 0.00000,C -180.00000} ; preinsert
  LIN {X -4624.998,Y -0.298,Z -43.502,A -90.00011,B 0.00000,C -180.00000} ; insert
  LIN {X -4624.998,Y -0.298,Z -43.502,A -90.00011,B 0.00000,C -180.00000} ; release
  LIN {X -4624.998,Y -0.298,Z 256.498,A -90.00011,B 0.00000,C -180.00000} ; retreat
  ; Step 2655, bar 173
  LIN {X -4499.998,Y -0.298,Z 1164.733,A -90.00011,B 0.00000,C -180.00000} ; outside
  LIN {X -4499.998,Y -0.298,Z 206.498,A -90.00011,B 0.00000,C -180.00000} ; preinsert
  LIN {X -4499.998,Y -0.298,Z -43.502,A -90.00011,B 0.00000,C -180.00000} ; insert
  LIN {X -4499.998,Y -0.298,Z -43.502,A -90.00011,B 0.00000,C -180.00000} ; release
  LIN {X -4499.998,Y -0.298,Z 256.498,A -90.00011,B 0.00000,C -180.00000} ; retreat
  ; Step 2656, bar 172
  LIN {X -4374.998,Y -0.298,Z 1164.733,A -90.00011,B 0.00000,C -180.00000} ; outside
  LIN {X -4374.998,Y -0.298,Z 206.498,A -90.00011,B 0.00000,C -180.00000} ; preinsert
  LIN {X -4374.998,Y -0.298,Z -43.502,A -90.00011,B 0.00000,C -180.00000} ; insert
  LIN {X -4374.998,Y -0.298,Z -43.502,A -90.00011,B 0.00000,C -180.00000} ; release
  LIN {X -4374.998,Y -0.298,Z 256.498,A -90.00011,B 0.00000,C -180.00000} ; retreat
  ; Step 2657, bar 171
  LIN {X -4249.998,Y -0.298,Z 1164.733,A -90.00011,B 0.00000,C -180.00000} ; outside
  LIN {X -4249.998,Y -0.298,Z 206.498,A -90.00011,B 0.00000,C -180.00000} ; preinsert
  LIN {X -4249.998,Y -0.298,Z -43.502,A -90.00011,B 0.00000,C -180.00000} ; insert
  LIN {X -4249.998,Y -0.298,Z -43.502,A -90.00011,B 0.00000,C -180.00000} ; release
  LIN {X -4249.998,Y -0.298,Z 256.498,A -90.00011,B 0.00000,C -180.00000} ; retreat
  ; Step 2658, bar 170
  LIN {X -4124.998,Y -0.298,Z 1164.733,A -90.00011,B 0.00000,C -180.00000} ; outside
  LIN {X -4124.998,Y -0.298,Z 206.498,A -90.00011,B 0.00000,C -180.00000} ; preinsert
  LIN {X -4124.998,Y -0.298,Z -43.502,A -90.00011,B 0.00000,C -180.00000} ; insert
  LIN {X -4124.998,Y -0.298,Z -43.502,A -90.00011,B 0.00000,C -180.00000} ; release
  LIN {X -4124.998,Y -0.298,Z 256.498,A -90.00011,B 0.00000,C -180.00000} ; retreat
  ; Step 2659, bar 169
  LIN {X -3999.998,Y -0.298,Z 1164.733,A -90.00011,B 0.00000,C -180.00000} ; outside
  LIN {X -3999.998,Y -0.298,Z 206.498,A -90.00011,B 0.00000,C -180.00000} ; preinsert
  LIN {X -3999.998,Y -0.298,Z -43.502,A -90.00011,B 0.00000,C -180.00000} ; insert
  LIN {X -3999.998,Y -0.298,Z -43.502,A -90.00011,B 0.00000,C -180.00000} ; release
  LIN {X -3999.998,Y -0.298,Z 256.498,A -90.00011,B 0.00000,C -180.00000} ; retreat
  ; Step 2660, bar 168
  LIN {X -3874.998,Y -0.298,Z 1164.733,A -90.00011,B 0.00000,C -180.00000} ; outside
  LIN {X -3874.998,Y -0.298,Z 206.498,A -90.00011,B 0.00000,C -180.00000} ; preinsert
  LIN {X -3874.998,Y -0.298,Z -43.502,A -90.00011,B 0.00000,C -180.00000} ; insert
  LIN {X -3874.998,Y -0.298,Z -43.502,A -90.00011,B 0.00000,C -180.00000} ; release
  LIN {X -3874.998,Y -0.298,Z 256.498,A -90.00011,B 0.00000,C -180.00000} ; retreat
  ; Step 2661, bar 167
  LIN {X -3749.998,Y -0.298,Z 1164.733,A -90.00011,B 0.00000,C -180.00000} ; outside
  LIN {X -3749.998,Y -0.298,Z 206.498,A -90.00011,B 0.00000,C -180.00000} ; preinsert
  LIN {X -3749.998,Y -0.298,Z -43.502,A -90.00011,B 0.00000,C -180.00000} ; insert
  LIN {X -3749.998,Y -0.298,Z -43.502,A -90.00011,B 0.00000,C -180.00000} ; release
  LIN {X -3749.998,Y -0.298,Z 256.498,A -90.00011,B 0.00000,C -180.00000} ; retreat
  ; Step 2662, bar 166
  LIN {X -3624.998,Y -0.298,Z 1164.733,A -90.00011,B 0.00000,C -180.00000} ; outside
  LIN {X -3624.998,Y -0.298,Z 206.498,A -90.00011,B 0.00000,C -180.00000} ; preinsert
  LIN {X -3624.998,Y -0.298,Z -43.502,A -90.00011,B 0.00000,C -180.00000} ; insert
  LIN {X -3624.998,Y -0.298,Z -43.502,A -90.00011,B 0.00000,C -180.00000} ; release
  LIN {X -3624.998,Y -0.298,Z 256.498,A -90.00011,B 0.00000,C -180.00000} ; retreat
  ; Step 2663, bar 165
  LIN {X -3499.998,Y -0.298,Z 1164.733,A -90.00011,B 0.00000,C -180.00000} ; outside
  LIN {X -3499.998,Y -0.298,Z 206.498,A -90.00011,B 0.00000,C -180.00000} ; preinsert
  LIN {X -3499.998,Y -0.298,Z -43.502,A -90.00011,B 0.00000,C -180.00000} ; insert
  LIN {X -3499.998,Y -0.298,Z -43.502,A -90.00011,B 0.00000,C -180.00000} ; release
  LIN {X -3499.998,Y -0.298,Z 256.498,A -90.00011,B 0.00000,C -180.00000} ; retreat
  ; Step 2664, bar 164
  LIN {X -3374.998,Y -0.298,Z 1164.733,A -90.00011,B 0.00000,C -180.00000} ; outside
  LIN {X -3374.998,Y -0.298,Z 206.498,A -90.00011,B 0.00000,C -180.00000} ; preinsert
  LIN {X -3374.998,Y -0.298,Z -43.502,A -90.00011,B 0.00000,C -180.00000} ; insert
  LIN {X -3374.998,Y -0.298,Z -43.502,A -90.00011,B 0.00000,C -180.00000} ; release
  LIN {X -3374.998,Y -0.298,Z 256.498,A -90.00011,B 0.00000,C -180.00000} ; retreat
  ; Step 2665, bar 163
  LIN {X -3249.998,Y -0.298,Z 1164.733,A -90.00011,B 0.00000,C -180.00000} ; outside
  LIN {X -3249.998,Y -0.298,Z 206.498,A -90.00011,B 0.00000,C -180.00000} ; preinsert
  LIN {X -3249.998,Y -0.298,Z -43.502,A -90.00011,B 0.00000,C -180.00000} ; insert
  LIN {X -3249.998,Y -0.298,Z -43.502,A -90.00011,B 0.00000,C -180.00000} ; release
  LIN {X -3249.998,Y -0.298,Z 256.498,A -90.00011,B 0.00000,C -180.00000} ; retreat
  ; Step 2666, bar 162
  LIN {X -3124.998,Y -0.298,Z 1164.733,A -90.00011,B 0.00000,C -180.00000} ; outside
  LIN {X -3124.998,Y -0.298,Z 206.498,A -90.00011,B 0.00000,C -180.00000} ; preinsert
  LIN {X -3124.998,Y -0.298,Z -43.502,A -90.00011,B 0.00000,C -180.00000} ; insert
  LIN {X -3124.998,Y -0.298,Z -43.502,A -90.00011,B 0.00000,C -180.00000} ; release
  LIN {X -3124.998,Y -0.298,Z 256.498,A -90.00011,B 0.00000,C -180.00000} ; retreat
  ; Step 2667, bar 161
  LIN {X -2999.998,Y -0.298,Z 1164.733,A -90.00011,B 0.00000,C -180.00000} ; outside
  LIN {X -2999.998,Y -0.298,Z 206.498,A -90.00011,B 0.00000,C -180.00000} ; preinsert
  LIN {X -2999.998,Y -0.298,Z -43.502,A -90.00011,B 0.00000,C -180.00000} ; insert
  LIN {X -2999.998,Y -0.298,Z -43.502,A -90.00011,B 0.00000,C -180.00000} ; release
  LIN {X -2999.998,Y -0.298,Z 256.498,A -90.00011,B 0.00000,C -180.00000} ; retreat
  ; Step 2668, bar 160
  LIN {X -2874.998,Y -0.298,Z 1164.733,A -90.00011,B 0.00000,C -180.00000} ; outside
  LIN {X -2874.998,Y -0.298,Z 206.498,A -90.00011,B 0.00000,C -180.00000} ; preinsert
  LIN {X -2874.998,Y -0.298,Z -43.502,A -90.00011,B 0.00000,C -180.00000} ; insert
  LIN {X -2874.998,Y -0.298,Z -43.502,A -90.00011,B 0.00000,C -180.00000} ; release
  LIN {X -2874.998,Y -0.298,Z 256.498,A -90.00011,B 0.00000,C -180.00000} ; retreat
  ; Step 2669, bar 159
  LIN {X -2749.998,Y -0.298,Z 1164.733,A -90.00011,B 0.00000,C -180.00000} ; outside
  LIN {X -2749.998,Y -0.298,Z 206.498,A -90.00011,B 0.00000,C -180.00000} ; preinsert
  LIN {X -2749.998,Y -0.298,Z -43.502,A -90.00011,B 0.00000,C -180.00000} ; insert
  LIN {X -2749.998,Y -0.298,Z -43.502,A -90.00011,B 0.00000,C -180.00000} ; release
  LIN {X -2749.998,Y -0.298,Z 256.498,A -90.00011,B 0.00000,C -180.00000} ; retreat
  ; Step 2670, bar 158
  LIN {X -2624.998,Y -0.298,Z 1164.733,A -90.00011,B 0.00000,C -180.00000} ; outside
  LIN {X -2624.998,Y -0.298,Z 206.498,A -90.00011,B 0.00000,C -180.00000} ; preinsert
  LIN {X -2624.998,Y -0.298,Z -43.502,A -90.00011,B 0.00000,C -180.00000} ; insert
  LIN {X -2624.998,Y -0.298,Z -43.502,A -90.00011,B 0.00000,C -180.00000} ; release
  LIN {X -2624.998,Y -0.298,Z 256.498,A -90.00011,B 0.00000,C -180.00000} ; retreat
  ; Step 2671, bar 157
  LIN {X -2499.998,Y -0.298,Z 1164.733,A -90.00011,B 0.00000,C -180.00000} ; outside
  LIN {X -2499.998,Y -0.298,Z 206.498,A -90.00011,B 0.00000,C -180.00000} ; preinsert
  LIN {X -2499.998,Y -0.298,Z -43.502,A -90.00011,B 0.00000,C -180.00000} ; insert
  LIN {X -2499.998,Y -0.298,Z -43.502,A -90.00011,B 0.00000,C -180.00000} ; release
  LIN {X -2499.998,Y -0.298,Z 256.498,A -90.00011,B 0.00000,C -180.00000} ; retreat
  ; Step 2672, bar 156
  LIN {X -2374.998,Y -0.298,Z 1164.733,A -90.00011,B 0.00000,C -180.00000} ; outside
  LIN {X -2374.998,Y -0.298,Z 206.498,A -90.00011,B 0.00000,C -180.00000} ; preinsert
  LIN {X -2374.998,Y -0.298,Z -43.502,A -90.00011,B 0.00000,C -180.00000} ; insert
  LIN {X -2374.998,Y -0.298,Z -43.502,A -90.00011,B 0.00000,C -180.00000} ; release
  LIN {X -2374.998,Y -0.298,Z 256.498,A -90.00011,B 0.00000,C -180.00000} ; retreat
  ; Step 2673, bar 155
  LIN {X -2249.998,Y -0.298,Z 1164.733,A -90.00011,B 0.00000,C -180.00000} ; outside
  LIN {X -2249.998,Y -0.298,Z 206.498,A -90.00011,B 0.00000,C -180.00000} ; preinsert
  LIN {X -2249.998,Y -0.298,Z -43.502,A -90.00011,B 0.00000,C -180.00000} ; insert
  LIN {X -2249.998,Y -0.298,Z -43.502,A -90.00011,B 0.00000,C -180.00000} ; release
  LIN {X -2249.998,Y -0.298,Z 256.498,A -90.00011,B 0.00000,C -180.00000} ; retreat
  ; Step 2674, bar 154
  LIN {X -2124.998,Y -0.298,Z 1164.733,A -90.00011,B 0.00000,C -180.00000} ; outside
  LIN {X -2124.998,Y -0.298,Z 206.498,A -90.00011,B 0.00000,C -180.00000} ; preinsert
  LIN {X -2124.998,Y -0.298,Z -43.502,A -90.00011,B 0.00000,C -180.00000} ; insert
  LIN {X -2124.998,Y -0.298,Z -43.502,A -90.00011,B 0.00000,C -180.00000} ; release
  LIN {X -2124.998,Y -0.298,Z 256.498,A -90.00011,B 0.00000,C -180.00000} ; retreat
  ; Step 2675, bar 153
  LIN {X -1874.998,Y -0.298,Z 1164.733,A -90.00011,B 0.00000,C -180.00000} ; outside
  LIN {X -1874.998,Y -0.298,Z 206.498,A -90.00011,B 0.00000,C -180.00000} ; preinsert
  LIN {X -1874.998,Y -0.298,Z -43.502,A -90.00011,B 0.00000,C -180.00000} ; insert
  LIN {X -1874.998,Y -0.298,Z -43.502,A -90.00011,B 0.00000,C -180.00000} ; release
  LIN {X -1874.998,Y -0.298,Z 256.498,A -90.00011,B 0.00000,C -180.00000} ; retreat
  ; Step 2676, bar 152
  LIN {X -1749.998,Y -0.298,Z 1164.733,A -90.00011,B 0.00000,C -180.00000} ; outside
  LIN {X -1749.998,Y -0.298,Z 206.498,A -90.00011,B 0.00000,C -180.00000} ; preinsert
  LIN {X -1749.998,Y -0.298,Z -43.502,A -90.00011,B 0.00000,C -180.00000} ; insert
  LIN {X -1749.998,Y -0.298,Z -43.502,A -90.00011,B 0.00000,C -180.00000} ; release
  LIN {X -1749.998,Y -0.298,Z 256.498,A -90.00011,B 0.00000,C -180.00000} ; retreat
  ; Step 2677, bar 151
  LIN {X -1624.998,Y -0.298,Z 1164.733,A -90.00011,B 0.00000,C -180.00000} ; outside
  LIN {X -1624.998,Y -0.298,Z 206.498,A -90.00011,B 0.00000,C -180.00000} ; preinsert
  LIN {X -1624.998,Y -0.298,Z -43.502,A -90.00011,B 0.00000,C -180.00000} ; insert
  LIN {X -1624.998,Y -0.298,Z -43.502,A -90.00011,B 0.00000,C -180.00000} ; release
  LIN {X -1624.998,Y -0.298,Z 256.498,A -90.00011,B 0.00000,C -180.00000} ; retreat
  ; Step 2678, bar 150
  LIN {X -1499.998,Y -0.298,Z 1164.733,A -90.00011,B 0.00000,C -180.00000} ; outside
  LIN {X -1499.998,Y -0.298,Z 206.498,A -90.00011,B 0.00000,C -180.00000} ; preinsert
  LIN {X -1499.998,Y -0.298,Z -43.502,A -90.00011,B 0.00000,C -180.00000} ; insert
  LIN {X -1499.998,Y -0.298,Z -43.502,A -90.00011,B 0.00000,C -180.00000} ; release
  LIN {X -1499.998,Y -0.298,Z 256.498,A -90.00011,B 0.00000,C -180.00000} ; retreat
  ; Step 2679, bar 149
  LIN {X -1374.998,Y -0.298,Z 1164.733,A -90.00011,B 0.00000,C -180.00000} ; outside
  LIN {X -1374.998,Y -0.298,Z 206.498,A -90.00011,B 0.00000,C -180.00000} ; preinsert
  LIN {X -1374.998,Y -0.298,Z -43.502,A -90.00011,B 0.00000,C -180.00000} ; insert
  LIN {X -1374.998,Y -0.298,Z -43.502,A -90.00011,B 0.00000,C -180.00000} ; release
  LIN {X -1374.998,Y -0.298,Z 256.498,A -90.00011,B 0.00000,C -180.00000} ; retreat
  ; Step 2680, bar 148
  LIN {X -1249.998,Y -0.298,Z 1164.733,A -90.00011,B 0.00000,C -180.00000} ; outside
  LIN {X -1249.998,Y -0.298,Z 206.498,A -90.00011,B 0.00000,C -180.00000} ; preinsert
  LIN {X -1249.998,Y -0.298,Z -43.502,A -90.00011,B 0.00000,C -180.00000} ; insert
  LIN {X -1249.998,Y -0.298,Z -43.502,A -90.00011,B 0.00000,C -180.00000} ; release
  LIN {X -1249.998,Y -0.298,Z 256.498,A -90.00011,B 0.00000,C -180.00000} ; retreat
  ; Step 2681, bar 147
  LIN {X -1124.998,Y -0.298,Z 1164.733,A -90.00011,B 0.00000,C -180.00000} ; outside
  LIN {X -1124.998,Y -0.298,Z 206.498,A -90.00011,B 0.00000,C -180.00000} ; preinsert
  LIN {X -1124.998,Y -0.298,Z -43.502,A -90.00011,B 0.00000,C -180.00000} ; insert
  LIN {X -1124.998,Y -0.298,Z -43.502,A -90.00011,B 0.00000,C -180.00000} ; release
  LIN {X -1124.998,Y -0.298,Z 256.498,A -90.00011,B 0.00000,C -180.00000} ; retreat
  ; Step 2682, bar 146
  LIN {X -999.998,Y -0.298,Z 1164.733,A -90.00011,B 0.00000,C -180.00000} ; outside
  LIN {X -999.998,Y -0.298,Z 206.498,A -90.00011,B 0.00000,C -180.00000} ; preinsert
  LIN {X -999.998,Y -0.298,Z -43.502,A -90.00011,B 0.00000,C -180.00000} ; insert
